// TIA Portal V17 export
// export: Created 2025-03-07T09:17:26.5341874Z, ExportSetting WithDefaults, DisplayName Totally Integrated Automation Portal, DisplayVersion V17 Update 8, DisplayName TIA Portal Openness, DisplayVersion V17 Update 8, DisplayName TIA Portal Version Control Interface, DisplayVersion V17, DisplayName SINAMICS Startdrive Advanced, DisplayVersion V17 SP2, DisplayName SINAMICS Startdrive G110M, G120, G120C, G120D, G120P, G115D, DisplayVersion V17 SP2, DisplayName SINAMICS Startdrive G130, G150, S120, S150, SINAMICS MV, S210, DisplayVersion V17 SP2, DisplayName STEP 7 Professional, DisplayVersion V17 Update 8, DisplayName SINUMERIK ONE STEP 7 Toolbox, DisplayVersion V17 Update 12, DisplayName SINUMERIK 840D sl STEP 7 Toolbox, DisplayVersion V17 Update 12, DisplayName STEP 7 Safety, DisplayVersion V17 Update 6, DisplayName WinCC Advanced, DisplayVersion V17 Update 8
FUNCTION "FC365_NCK_M_CH7_UNIT_2_STA_4" : Void   // FC365, LAD
TITLE = Channel 1 data
{ S7_Optimized_Access := 'FALSE' }
AUTHOR : ETXETAR
VERSION : 1.0
// stored: AutoNumber false, IsIECCheckEnabled false, SetENOAutomatically false, UDAEnableTagReadback false
   VAR_TEMP
      auxm3 : Bool;
      auxm5 : Bool;
   END_VAR
   VAR_TEMP   // added for the SCL form of the ladder/FBD networks
      _w1 : Bool;
      _w2 : Bool;
   END_VAR
BEGIN

REGION Network 1: CALL FB331 M CODE EXTENDED CH4 / M CODE EXTENDED CHANNEL 2
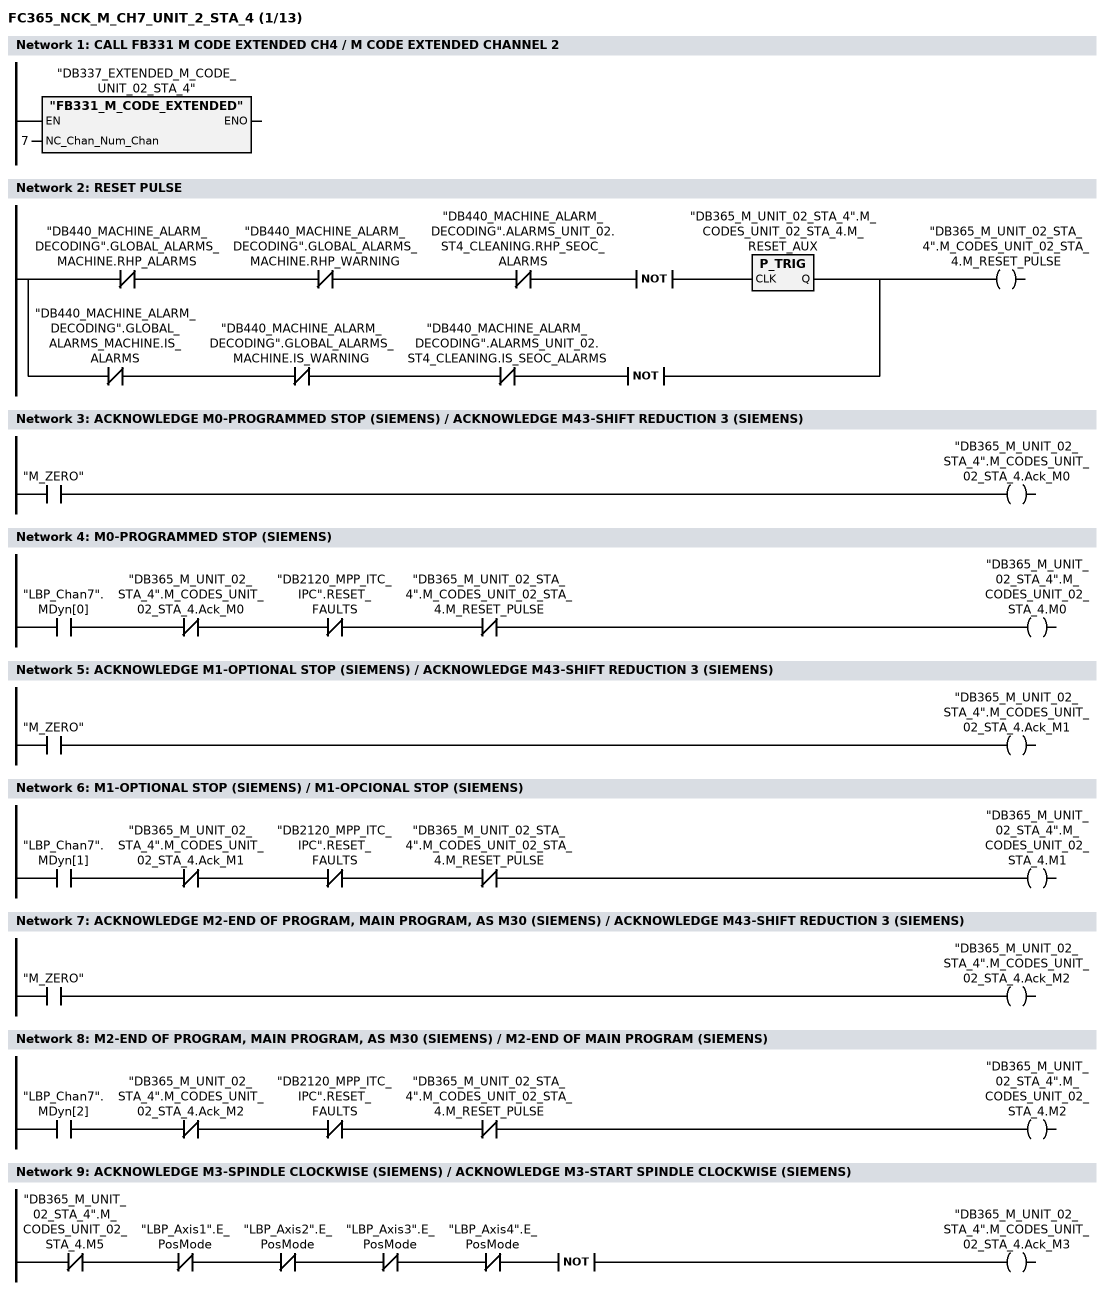
   RUNG wire#powerrail
      "DB337_EXTENDED_M_CODE_UNIT_02_STA_4"(NC_Chan_Num_Chan := 7)
   END_RUNG
   // the same network as SCL:
   "DB337_EXTENDED_M_CODE_UNIT_02_STA_4"(NC_Chan_Num_Chan := 7);   // "FB331_M_CODE_EXTENDED"
END_REGION

REGION Network 2: RESET PULSE
   RUNG wire#powerrail
      I_Contact( "DB440_MACHINE_ALARM_DECODING".GLOBAL_ALARMS_MACHINE.RHP_ALARMS )
      I_Contact( "DB440_MACHINE_ALARM_DECODING".GLOBAL_ALARMS_MACHINE.RHP_WARNING )
      I_Contact( "DB440_MACHINE_ALARM_DECODING".ALARMS_UNIT_02.ST4_CLEANING.RHP_SEOC_ALARMS )
      Not()
      P_Trig( "DB365_M_UNIT_02_STA_4".M_CODES_UNIT_02_STA_4.M_RESET_AUX )
      wire#w1
      Coil( "DB365_M_UNIT_02_STA_4".M_CODES_UNIT_02_STA_4.M_RESET_PULSE )
   END_RUNG
   RUNG wire#powerrail
      I_Contact( "DB440_MACHINE_ALARM_DECODING".GLOBAL_ALARMS_MACHINE.IS_ALARMS )
      I_Contact( "DB440_MACHINE_ALARM_DECODING".GLOBAL_ALARMS_MACHINE.IS_WARNING )
      I_Contact( "DB440_MACHINE_ALARM_DECODING".ALARMS_UNIT_02.ST4_CLEANING.IS_SEOC_ALARMS )
      Not()
   END_RUNG wire#w1
   // the same network as SCL:
   #_w1 := NOT (NOT "DB440_MACHINE_ALARM_DECODING".GLOBAL_ALARMS_MACHINE.RHP_ALARMS AND NOT "DB440_MACHINE_ALARM_DECODING".GLOBAL_ALARMS_MACHINE.RHP_WARNING AND NOT "DB440_MACHINE_ALARM_DECODING".ALARMS_UNIT_02.ST4_CLEANING.RHP_SEOC_ALARMS);
   #_w2 := #_w1 AND NOT "DB365_M_UNIT_02_STA_4".M_CODES_UNIT_02_STA_4.M_RESET_AUX;   // rising edge
   "DB365_M_UNIT_02_STA_4".M_CODES_UNIT_02_STA_4.M_RESET_AUX := #_w1;
   "DB365_M_UNIT_02_STA_4".M_CODES_UNIT_02_STA_4.M_RESET_PULSE := #_w2 OR NOT (NOT "DB440_MACHINE_ALARM_DECODING".GLOBAL_ALARMS_MACHINE.IS_ALARMS AND NOT "DB440_MACHINE_ALARM_DECODING".GLOBAL_ALARMS_MACHINE.IS_WARNING AND NOT "DB440_MACHINE_ALARM_DECODING".ALARMS_UNIT_02.ST4_CLEANING.IS_SEOC_ALARMS);
END_REGION

REGION Network 3: ACKNOWLEDGE M0-PROGRAMMED STOP (SIEMENS) / ACKNOWLEDGE M43-SHIFT REDUCTION 3 (SIEMENS)
   RUNG wire#powerrail
      Contact( "M_ZERO" )
      Coil( "DB365_M_UNIT_02_STA_4".M_CODES_UNIT_02_STA_4.Ack_M0 )
   END_RUNG
   // the same network as SCL:
   "DB365_M_UNIT_02_STA_4".M_CODES_UNIT_02_STA_4.Ack_M0 := "M_ZERO";
END_REGION

REGION Network 4: M0-PROGRAMMED STOP (SIEMENS)
   RUNG wire#powerrail
      Contact( "LBP_Chan7".MDyn[0] )
      I_Contact( "DB365_M_UNIT_02_STA_4".M_CODES_UNIT_02_STA_4.Ack_M0 )
      I_Contact( "DB2120_MPP_ITC_IPC".RESET_FAULTS )
      I_Contact( "DB365_M_UNIT_02_STA_4".M_CODES_UNIT_02_STA_4.M_RESET_PULSE )
      Coil( "DB365_M_UNIT_02_STA_4".M_CODES_UNIT_02_STA_4.M0 )
   END_RUNG
   // the same network as SCL:
   "DB365_M_UNIT_02_STA_4".M_CODES_UNIT_02_STA_4.M0 := "LBP_Chan7".MDyn[0] AND NOT "DB365_M_UNIT_02_STA_4".M_CODES_UNIT_02_STA_4.Ack_M0 AND NOT "DB2120_MPP_ITC_IPC".RESET_FAULTS AND NOT "DB365_M_UNIT_02_STA_4".M_CODES_UNIT_02_STA_4.M_RESET_PULSE;
END_REGION

REGION Network 5: ACKNOWLEDGE M1-OPTIONAL STOP (SIEMENS) / ACKNOWLEDGE M43-SHIFT REDUCTION 3 (SIEMENS)
   RUNG wire#powerrail
      Contact( "M_ZERO" )
      Coil( "DB365_M_UNIT_02_STA_4".M_CODES_UNIT_02_STA_4.Ack_M1 )
   END_RUNG
   // the same network as SCL:
   "DB365_M_UNIT_02_STA_4".M_CODES_UNIT_02_STA_4.Ack_M1 := "M_ZERO";
END_REGION

REGION Network 6: M1-OPTIONAL STOP (SIEMENS) / M1-OPCIONAL STOP (SIEMENS)
   RUNG wire#powerrail
      Contact( "LBP_Chan7".MDyn[1] )
      I_Contact( "DB365_M_UNIT_02_STA_4".M_CODES_UNIT_02_STA_4.Ack_M1 )
      I_Contact( "DB2120_MPP_ITC_IPC".RESET_FAULTS )
      I_Contact( "DB365_M_UNIT_02_STA_4".M_CODES_UNIT_02_STA_4.M_RESET_PULSE )
      Coil( "DB365_M_UNIT_02_STA_4".M_CODES_UNIT_02_STA_4.M1 )
   END_RUNG
   // the same network as SCL:
   "DB365_M_UNIT_02_STA_4".M_CODES_UNIT_02_STA_4.M1 := "LBP_Chan7".MDyn[1] AND NOT "DB365_M_UNIT_02_STA_4".M_CODES_UNIT_02_STA_4.Ack_M1 AND NOT "DB2120_MPP_ITC_IPC".RESET_FAULTS AND NOT "DB365_M_UNIT_02_STA_4".M_CODES_UNIT_02_STA_4.M_RESET_PULSE;
END_REGION

REGION Network 7: ACKNOWLEDGE M2-END OF PROGRAM, MAIN PROGRAM, AS M30 (SIEMENS) / ACKNOWLEDGE M43-SHIFT REDUCTION 3 (SIEMENS)
   RUNG wire#powerrail
      Contact( "M_ZERO" )
      Coil( "DB365_M_UNIT_02_STA_4".M_CODES_UNIT_02_STA_4.Ack_M2 )
   END_RUNG
   // the same network as SCL:
   "DB365_M_UNIT_02_STA_4".M_CODES_UNIT_02_STA_4.Ack_M2 := "M_ZERO";
END_REGION

REGION Network 8: M2-END OF PROGRAM, MAIN PROGRAM, AS M30 (SIEMENS) / M2-END OF MAIN PROGRAM (SIEMENS)
   RUNG wire#powerrail
      Contact( "LBP_Chan7".MDyn[2] )
      I_Contact( "DB365_M_UNIT_02_STA_4".M_CODES_UNIT_02_STA_4.Ack_M2 )
      I_Contact( "DB2120_MPP_ITC_IPC".RESET_FAULTS )
      I_Contact( "DB365_M_UNIT_02_STA_4".M_CODES_UNIT_02_STA_4.M_RESET_PULSE )
      Coil( "DB365_M_UNIT_02_STA_4".M_CODES_UNIT_02_STA_4.M2 )
   END_RUNG
   // the same network as SCL:
   "DB365_M_UNIT_02_STA_4".M_CODES_UNIT_02_STA_4.M2 := "LBP_Chan7".MDyn[2] AND NOT "DB365_M_UNIT_02_STA_4".M_CODES_UNIT_02_STA_4.Ack_M2 AND NOT "DB2120_MPP_ITC_IPC".RESET_FAULTS AND NOT "DB365_M_UNIT_02_STA_4".M_CODES_UNIT_02_STA_4.M_RESET_PULSE;
END_REGION

REGION Network 9: ACKNOWLEDGE M3-SPINDLE CLOCKWISE (SIEMENS) / ACKNOWLEDGE M3-START SPINDLE CLOCKWISE (SIEMENS)
   RUNG wire#powerrail
      I_Contact( "DB365_M_UNIT_02_STA_4".M_CODES_UNIT_02_STA_4.M5 )
      I_Contact( "LBP_Axis1".E_PosMode )
      I_Contact( "LBP_Axis2".E_PosMode )
      I_Contact( "LBP_Axis3".E_PosMode )
      I_Contact( "LBP_Axis4".E_PosMode )
      Not()
      Coil( "DB365_M_UNIT_02_STA_4".M_CODES_UNIT_02_STA_4.Ack_M3 )
   END_RUNG
   // the same network as SCL:
   "DB365_M_UNIT_02_STA_4".M_CODES_UNIT_02_STA_4.Ack_M3 := NOT (NOT "DB365_M_UNIT_02_STA_4".M_CODES_UNIT_02_STA_4.M5 AND NOT "LBP_Axis1".E_PosMode AND NOT "LBP_Axis2".E_PosMode AND NOT "LBP_Axis3".E_PosMode AND NOT "LBP_Axis4".E_PosMode);
END_REGION

REGION Network 10: M3-SPINDLE CLOCKWISE AUXILIARY (SIEMENS) / Extended address M function 1 (16 bit INT)
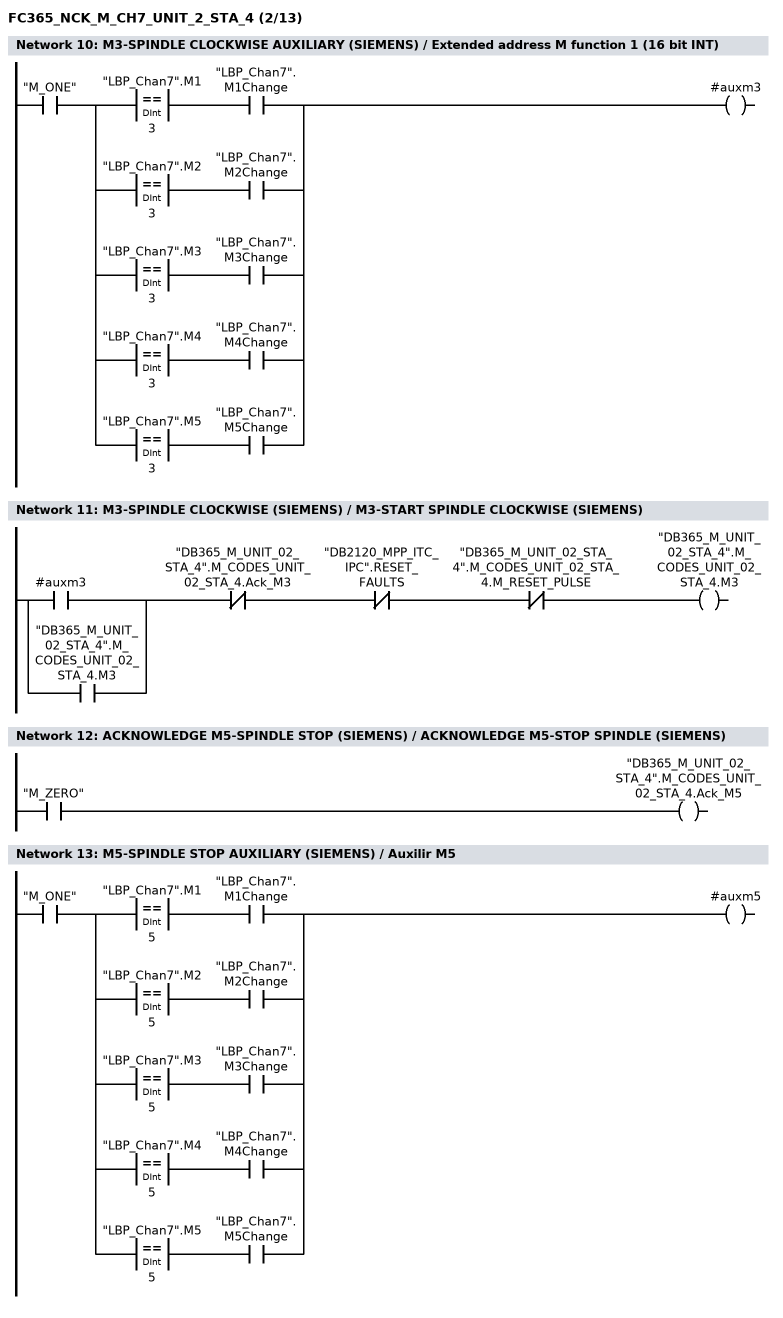
   RUNG wire#powerrail
      Contact( "M_ONE" )
      wire#w1
      { S7_Templates := "SrcType := DInt" } EQ_Contact(in1 := "LBP_Chan7".M1, in2 := 3)
      Contact( "LBP_Chan7".M1Change )
      wire#w2
      Coil( #auxm3 )
   END_RUNG
   RUNG wire#w1
      { S7_Templates := "SrcType := DInt" } EQ_Contact(in1 := "LBP_Chan7".M2, in2 := 3)
      Contact( "LBP_Chan7".M2Change )
   END_RUNG wire#w2
   RUNG wire#w1
      { S7_Templates := "SrcType := DInt" } EQ_Contact(in1 := "LBP_Chan7".M3, in2 := 3)
      Contact( "LBP_Chan7".M3Change )
   END_RUNG wire#w2
   RUNG wire#w1
      { S7_Templates := "SrcType := DInt" } EQ_Contact(in1 := "LBP_Chan7".M4, in2 := 3)
      Contact( "LBP_Chan7".M4Change )
   END_RUNG wire#w2
   RUNG wire#w1
      { S7_Templates := "SrcType := DInt" } EQ_Contact(in1 := "LBP_Chan7".M5, in2 := 3)
      Contact( "LBP_Chan7".M5Change )
   END_RUNG wire#w2
   // the same network as SCL:
   #auxm3 := "M_ONE" AND ((("LBP_Chan7".M1 = 3) AND "LBP_Chan7".M1Change) OR (("LBP_Chan7".M2 = 3) AND "LBP_Chan7".M2Change) OR (("LBP_Chan7".M3 = 3) AND "LBP_Chan7".M3Change) OR (("LBP_Chan7".M4 = 3) AND "LBP_Chan7".M4Change) OR (("LBP_Chan7".M5 = 3) AND "LBP_Chan7".M5Change));
END_REGION

REGION Network 11: M3-SPINDLE CLOCKWISE (SIEMENS) / M3-START SPINDLE CLOCKWISE (SIEMENS)
   RUNG wire#powerrail
      Contact( #auxm3 )
      wire#w1
      I_Contact( "DB365_M_UNIT_02_STA_4".M_CODES_UNIT_02_STA_4.Ack_M3 )
      I_Contact( "DB2120_MPP_ITC_IPC".RESET_FAULTS )
      I_Contact( "DB365_M_UNIT_02_STA_4".M_CODES_UNIT_02_STA_4.M_RESET_PULSE )
      Coil( "DB365_M_UNIT_02_STA_4".M_CODES_UNIT_02_STA_4.M3 )
   END_RUNG
   RUNG wire#powerrail
      Contact( "DB365_M_UNIT_02_STA_4".M_CODES_UNIT_02_STA_4.M3 )
   END_RUNG wire#w1
   // the same network as SCL:
   "DB365_M_UNIT_02_STA_4".M_CODES_UNIT_02_STA_4.M3 := (#auxm3 OR "DB365_M_UNIT_02_STA_4".M_CODES_UNIT_02_STA_4.M3) AND NOT "DB365_M_UNIT_02_STA_4".M_CODES_UNIT_02_STA_4.Ack_M3 AND NOT "DB2120_MPP_ITC_IPC".RESET_FAULTS AND NOT "DB365_M_UNIT_02_STA_4".M_CODES_UNIT_02_STA_4.M_RESET_PULSE;
END_REGION

REGION Network 12: ACKNOWLEDGE M5-SPINDLE STOP (SIEMENS) / ACKNOWLEDGE M5-STOP SPINDLE (SIEMENS)
   RUNG wire#powerrail
      Contact( "M_ZERO" )
      Coil( "DB365_M_UNIT_02_STA_4".M_CODES_UNIT_02_STA_4.Ack_M5 )
   END_RUNG
   // the same network as SCL:
   "DB365_M_UNIT_02_STA_4".M_CODES_UNIT_02_STA_4.Ack_M5 := "M_ZERO";
END_REGION

REGION Network 13: M5-SPINDLE STOP AUXILIARY (SIEMENS) / Auxilir M5
   RUNG wire#powerrail
      Contact( "M_ONE" )
      wire#w1
      { S7_Templates := "SrcType := DInt" } EQ_Contact(in1 := "LBP_Chan7".M1, in2 := 5)
      Contact( "LBP_Chan7".M1Change )
      wire#w2
      Coil( #auxm5 )
   END_RUNG
   RUNG wire#w1
      { S7_Templates := "SrcType := DInt" } EQ_Contact(in1 := "LBP_Chan7".M2, in2 := 5)
      Contact( "LBP_Chan7".M2Change )
   END_RUNG wire#w2
   RUNG wire#w1
      { S7_Templates := "SrcType := DInt" } EQ_Contact(in1 := "LBP_Chan7".M3, in2 := 5)
      Contact( "LBP_Chan7".M3Change )
   END_RUNG wire#w2
   RUNG wire#w1
      { S7_Templates := "SrcType := DInt" } EQ_Contact(in1 := "LBP_Chan7".M4, in2 := 5)
      Contact( "LBP_Chan7".M4Change )
   END_RUNG wire#w2
   RUNG wire#w1
      { S7_Templates := "SrcType := DInt" } EQ_Contact(in1 := "LBP_Chan7".M5, in2 := 5)
      Contact( "LBP_Chan7".M5Change )
   END_RUNG wire#w2
   // the same network as SCL:
   #auxm5 := "M_ONE" AND ((("LBP_Chan7".M1 = 5) AND "LBP_Chan7".M1Change) OR (("LBP_Chan7".M2 = 5) AND "LBP_Chan7".M2Change) OR (("LBP_Chan7".M3 = 5) AND "LBP_Chan7".M3Change) OR (("LBP_Chan7".M4 = 5) AND "LBP_Chan7".M4Change) OR (("LBP_Chan7".M5 = 5) AND "LBP_Chan7".M5Change));
END_REGION

REGION Network 14: M5-SPINDLE STOP (SIEMENS) / M5-STOP SPINDLE (SIEMENS)
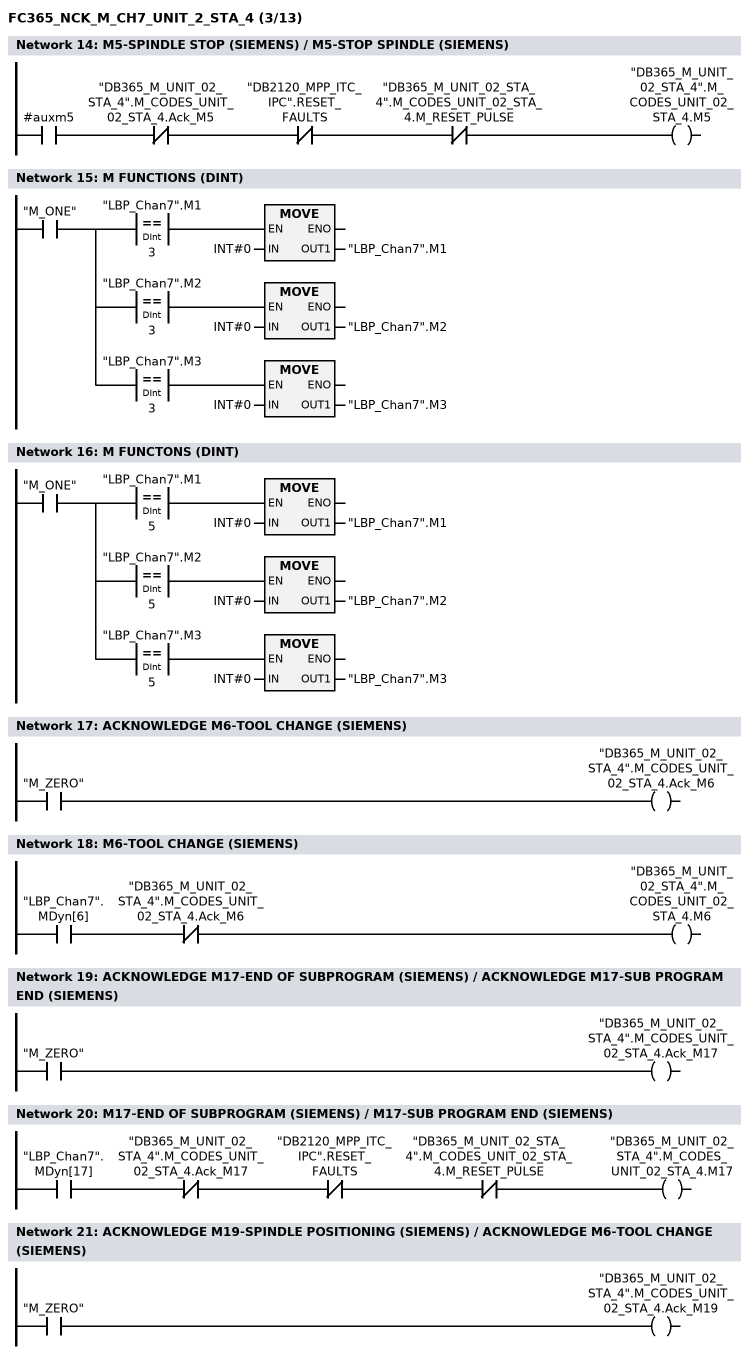
   RUNG wire#powerrail
      Contact( #auxm5 )
      I_Contact( "DB365_M_UNIT_02_STA_4".M_CODES_UNIT_02_STA_4.Ack_M5 )
      I_Contact( "DB2120_MPP_ITC_IPC".RESET_FAULTS )
      I_Contact( "DB365_M_UNIT_02_STA_4".M_CODES_UNIT_02_STA_4.M_RESET_PULSE )
      Coil( "DB365_M_UNIT_02_STA_4".M_CODES_UNIT_02_STA_4.M5 )
   END_RUNG
   // the same network as SCL:
   "DB365_M_UNIT_02_STA_4".M_CODES_UNIT_02_STA_4.M5 := #auxm5 AND NOT "DB365_M_UNIT_02_STA_4".M_CODES_UNIT_02_STA_4.Ack_M5 AND NOT "DB2120_MPP_ITC_IPC".RESET_FAULTS AND NOT "DB365_M_UNIT_02_STA_4".M_CODES_UNIT_02_STA_4.M_RESET_PULSE;
END_REGION

REGION Network 15: M FUNCTIONS (DINT)
   RUNG wire#powerrail
      Contact( "M_ONE" )
      wire#w1
      { S7_Templates := "SrcType := DInt" } EQ_Contact(in1 := "LBP_Chan7".M1, in2 := 3)
      { S7_GenerateENO := "TRUE" } Move(in := INT#0, out1 => "LBP_Chan7".M1)
   END_RUNG
   RUNG wire#w1
      { S7_Templates := "SrcType := DInt" } EQ_Contact(in1 := "LBP_Chan7".M2, in2 := 3)
      { S7_GenerateENO := "TRUE" } Move(in := INT#0, out1 => "LBP_Chan7".M2)
   END_RUNG
   RUNG wire#w1
      { S7_Templates := "SrcType := DInt" } EQ_Contact(in1 := "LBP_Chan7".M3, in2 := 3)
      { S7_GenerateENO := "TRUE" } Move(in := INT#0, out1 => "LBP_Chan7".M3)
   END_RUNG
   // the same network as SCL:
   IF "M_ONE" AND ("LBP_Chan7".M1 = 3) THEN "LBP_Chan7".M1 := INT#0; END_IF;
   IF "M_ONE" AND ("LBP_Chan7".M2 = 3) THEN "LBP_Chan7".M2 := INT#0; END_IF;
   IF "M_ONE" AND ("LBP_Chan7".M3 = 3) THEN "LBP_Chan7".M3 := INT#0; END_IF;
END_REGION

REGION Network 16: M FUNCTONS (DINT)
   RUNG wire#powerrail
      Contact( "M_ONE" )
      wire#w1
      { S7_Templates := "SrcType := DInt" } EQ_Contact(in1 := "LBP_Chan7".M1, in2 := 5)
      { S7_GenerateENO := "TRUE" } Move(in := INT#0, out1 => "LBP_Chan7".M1)
   END_RUNG
   RUNG wire#w1
      { S7_Templates := "SrcType := DInt" } EQ_Contact(in1 := "LBP_Chan7".M2, in2 := 5)
      { S7_GenerateENO := "TRUE" } Move(in := INT#0, out1 => "LBP_Chan7".M2)
   END_RUNG
   RUNG wire#w1
      { S7_Templates := "SrcType := DInt" } EQ_Contact(in1 := "LBP_Chan7".M3, in2 := 5)
      { S7_GenerateENO := "TRUE" } Move(in := INT#0, out1 => "LBP_Chan7".M3)
   END_RUNG
   // the same network as SCL:
   IF "M_ONE" AND ("LBP_Chan7".M1 = 5) THEN "LBP_Chan7".M1 := INT#0; END_IF;
   IF "M_ONE" AND ("LBP_Chan7".M2 = 5) THEN "LBP_Chan7".M2 := INT#0; END_IF;
   IF "M_ONE" AND ("LBP_Chan7".M3 = 5) THEN "LBP_Chan7".M3 := INT#0; END_IF;
END_REGION

REGION Network 17: ACKNOWLEDGE M6-TOOL CHANGE (SIEMENS)
   RUNG wire#powerrail
      Contact( "M_ZERO" )
      Coil( "DB365_M_UNIT_02_STA_4".M_CODES_UNIT_02_STA_4.Ack_M6 )
   END_RUNG
   // the same network as SCL:
   "DB365_M_UNIT_02_STA_4".M_CODES_UNIT_02_STA_4.Ack_M6 := "M_ZERO";
END_REGION

REGION Network 18: M6-TOOL CHANGE (SIEMENS)
   RUNG wire#powerrail
      Contact( "LBP_Chan7".MDyn[6] )
      I_Contact( "DB365_M_UNIT_02_STA_4".M_CODES_UNIT_02_STA_4.Ack_M6 )
      Coil( "DB365_M_UNIT_02_STA_4".M_CODES_UNIT_02_STA_4.M6 )
   END_RUNG
   // the same network as SCL:
   "DB365_M_UNIT_02_STA_4".M_CODES_UNIT_02_STA_4.M6 := "LBP_Chan7".MDyn[6] AND NOT "DB365_M_UNIT_02_STA_4".M_CODES_UNIT_02_STA_4.Ack_M6;
END_REGION

REGION Network 19: ACKNOWLEDGE M17-END OF SUBPROGRAM (SIEMENS) / ACKNOWLEDGE M17-SUB PROGRAM END (SIEMENS)
   RUNG wire#powerrail
      Contact( "M_ZERO" )
      Coil( "DB365_M_UNIT_02_STA_4".M_CODES_UNIT_02_STA_4.Ack_M17 )
   END_RUNG
   // the same network as SCL:
   "DB365_M_UNIT_02_STA_4".M_CODES_UNIT_02_STA_4.Ack_M17 := "M_ZERO";
END_REGION

REGION Network 20: M17-END OF SUBPROGRAM (SIEMENS) / M17-SUB PROGRAM END (SIEMENS)
   RUNG wire#powerrail
      Contact( "LBP_Chan7".MDyn[17] )
      I_Contact( "DB365_M_UNIT_02_STA_4".M_CODES_UNIT_02_STA_4.Ack_M17 )
      I_Contact( "DB2120_MPP_ITC_IPC".RESET_FAULTS )
      I_Contact( "DB365_M_UNIT_02_STA_4".M_CODES_UNIT_02_STA_4.M_RESET_PULSE )
      Coil( "DB365_M_UNIT_02_STA_4".M_CODES_UNIT_02_STA_4.M17 )
   END_RUNG
   // the same network as SCL:
   "DB365_M_UNIT_02_STA_4".M_CODES_UNIT_02_STA_4.M17 := "LBP_Chan7".MDyn[17] AND NOT "DB365_M_UNIT_02_STA_4".M_CODES_UNIT_02_STA_4.Ack_M17 AND NOT "DB2120_MPP_ITC_IPC".RESET_FAULTS AND NOT "DB365_M_UNIT_02_STA_4".M_CODES_UNIT_02_STA_4.M_RESET_PULSE;
END_REGION

REGION Network 21: ACKNOWLEDGE M19-SPINDLE POSITIONING (SIEMENS) / ACKNOWLEDGE M6-TOOL CHANGE (SIEMENS)
   RUNG wire#powerrail
      Contact( "M_ZERO" )
      Coil( "DB365_M_UNIT_02_STA_4".M_CODES_UNIT_02_STA_4.Ack_M19 )
   END_RUNG
   // the same network as SCL:
   "DB365_M_UNIT_02_STA_4".M_CODES_UNIT_02_STA_4.Ack_M19 := "M_ZERO";
END_REGION

REGION Network 22: M19-SPINDLE POSITIONING (SIEMENS) / M6-TOOL CHANGE (SIEMENS)
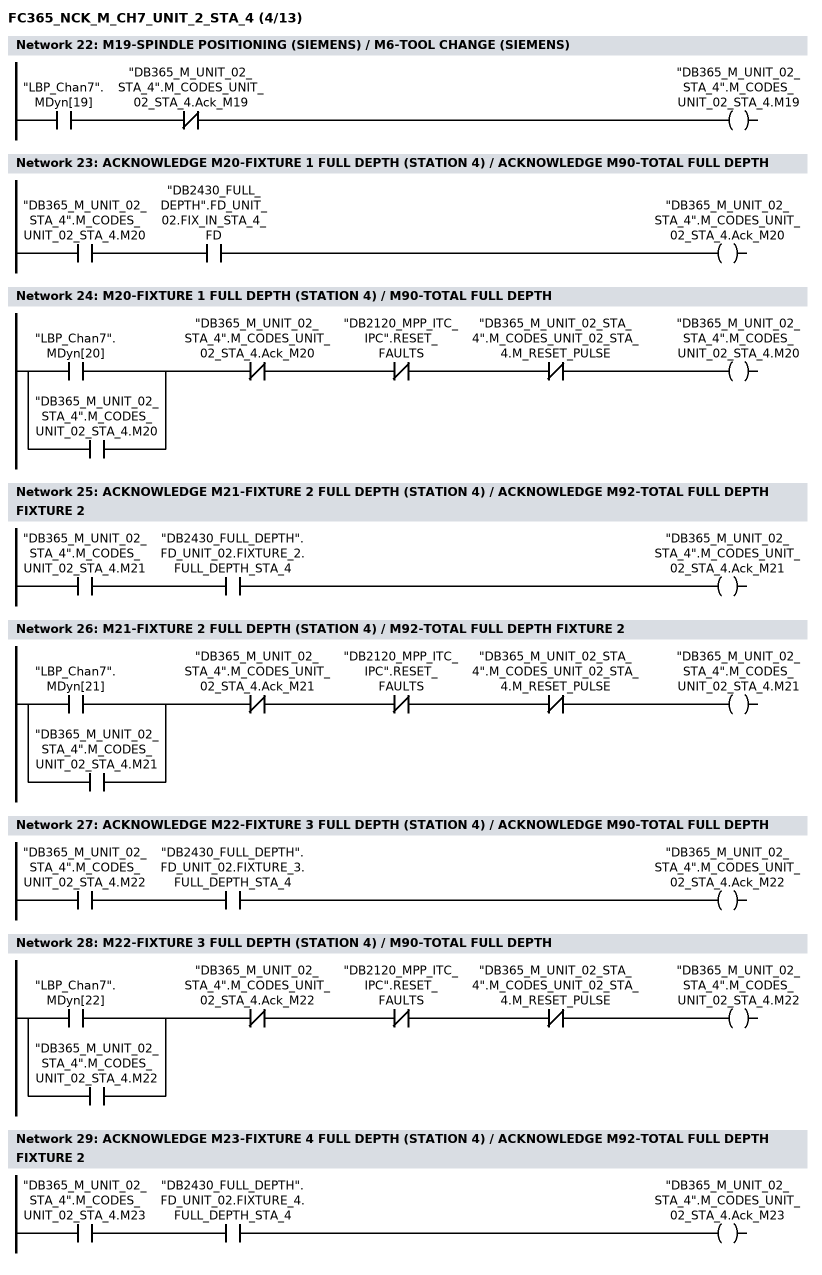
   RUNG wire#powerrail
      Contact( "LBP_Chan7".MDyn[19] )
      I_Contact( "DB365_M_UNIT_02_STA_4".M_CODES_UNIT_02_STA_4.Ack_M19 )
      Coil( "DB365_M_UNIT_02_STA_4".M_CODES_UNIT_02_STA_4.M19 )
   END_RUNG
   // the same network as SCL:
   "DB365_M_UNIT_02_STA_4".M_CODES_UNIT_02_STA_4.M19 := "LBP_Chan7".MDyn[19] AND NOT "DB365_M_UNIT_02_STA_4".M_CODES_UNIT_02_STA_4.Ack_M19;
END_REGION

REGION Network 23: ACKNOWLEDGE M20-FIXTURE 1 FULL DEPTH (STATION 4) / ACKNOWLEDGE M90-TOTAL FULL DEPTH
   RUNG wire#powerrail
      Contact( "DB365_M_UNIT_02_STA_4".M_CODES_UNIT_02_STA_4.M20 )
      Contact( "DB2430_FULL_DEPTH".FD_UNIT_02.FIX_IN_STA_4_FD )
      Coil( "DB365_M_UNIT_02_STA_4".M_CODES_UNIT_02_STA_4.Ack_M20 )
   END_RUNG
   // the same network as SCL:
   "DB365_M_UNIT_02_STA_4".M_CODES_UNIT_02_STA_4.Ack_M20 := "DB365_M_UNIT_02_STA_4".M_CODES_UNIT_02_STA_4.M20 AND "DB2430_FULL_DEPTH".FD_UNIT_02.FIX_IN_STA_4_FD;
END_REGION

REGION Network 24: M20-FIXTURE 1 FULL DEPTH (STATION 4) / M90-TOTAL FULL DEPTH
   RUNG wire#powerrail
      Contact( "LBP_Chan7".MDyn[20] )
      wire#w1
      I_Contact( "DB365_M_UNIT_02_STA_4".M_CODES_UNIT_02_STA_4.Ack_M20 )
      I_Contact( "DB2120_MPP_ITC_IPC".RESET_FAULTS )
      I_Contact( "DB365_M_UNIT_02_STA_4".M_CODES_UNIT_02_STA_4.M_RESET_PULSE )
      Coil( "DB365_M_UNIT_02_STA_4".M_CODES_UNIT_02_STA_4.M20 )
   END_RUNG
   RUNG wire#powerrail
      Contact( "DB365_M_UNIT_02_STA_4".M_CODES_UNIT_02_STA_4.M20 )
   END_RUNG wire#w1
   // the same network as SCL:
   "DB365_M_UNIT_02_STA_4".M_CODES_UNIT_02_STA_4.M20 := ("LBP_Chan7".MDyn[20] OR "DB365_M_UNIT_02_STA_4".M_CODES_UNIT_02_STA_4.M20) AND NOT "DB365_M_UNIT_02_STA_4".M_CODES_UNIT_02_STA_4.Ack_M20 AND NOT "DB2120_MPP_ITC_IPC".RESET_FAULTS AND NOT "DB365_M_UNIT_02_STA_4".M_CODES_UNIT_02_STA_4.M_RESET_PULSE;
END_REGION

REGION Network 25: ACKNOWLEDGE M21-FIXTURE 2 FULL DEPTH (STATION 4) / ACKNOWLEDGE M92-TOTAL FULL DEPTH FIXTURE 2
   RUNG wire#powerrail
      Contact( "DB365_M_UNIT_02_STA_4".M_CODES_UNIT_02_STA_4.M21 )
      Contact( "DB2430_FULL_DEPTH".FD_UNIT_02.FIXTURE_2.FULL_DEPTH_STA_4 )
      Coil( "DB365_M_UNIT_02_STA_4".M_CODES_UNIT_02_STA_4.Ack_M21 )
   END_RUNG
   // the same network as SCL:
   "DB365_M_UNIT_02_STA_4".M_CODES_UNIT_02_STA_4.Ack_M21 := "DB365_M_UNIT_02_STA_4".M_CODES_UNIT_02_STA_4.M21 AND "DB2430_FULL_DEPTH".FD_UNIT_02.FIXTURE_2.FULL_DEPTH_STA_4;
END_REGION

REGION Network 26: M21-FIXTURE 2 FULL DEPTH (STATION 4) / M92-TOTAL FULL DEPTH FIXTURE 2
   RUNG wire#powerrail
      Contact( "LBP_Chan7".MDyn[21] )
      wire#w1
      I_Contact( "DB365_M_UNIT_02_STA_4".M_CODES_UNIT_02_STA_4.Ack_M21 )
      I_Contact( "DB2120_MPP_ITC_IPC".RESET_FAULTS )
      I_Contact( "DB365_M_UNIT_02_STA_4".M_CODES_UNIT_02_STA_4.M_RESET_PULSE )
      Coil( "DB365_M_UNIT_02_STA_4".M_CODES_UNIT_02_STA_4.M21 )
   END_RUNG
   RUNG wire#powerrail
      Contact( "DB365_M_UNIT_02_STA_4".M_CODES_UNIT_02_STA_4.M21 )
   END_RUNG wire#w1
   // the same network as SCL:
   "DB365_M_UNIT_02_STA_4".M_CODES_UNIT_02_STA_4.M21 := ("LBP_Chan7".MDyn[21] OR "DB365_M_UNIT_02_STA_4".M_CODES_UNIT_02_STA_4.M21) AND NOT "DB365_M_UNIT_02_STA_4".M_CODES_UNIT_02_STA_4.Ack_M21 AND NOT "DB2120_MPP_ITC_IPC".RESET_FAULTS AND NOT "DB365_M_UNIT_02_STA_4".M_CODES_UNIT_02_STA_4.M_RESET_PULSE;
END_REGION

REGION Network 27: ACKNOWLEDGE M22-FIXTURE 3 FULL DEPTH (STATION 4) / ACKNOWLEDGE M90-TOTAL FULL DEPTH
   RUNG wire#powerrail
      Contact( "DB365_M_UNIT_02_STA_4".M_CODES_UNIT_02_STA_4.M22 )
      Contact( "DB2430_FULL_DEPTH".FD_UNIT_02.FIXTURE_3.FULL_DEPTH_STA_4 )
      Coil( "DB365_M_UNIT_02_STA_4".M_CODES_UNIT_02_STA_4.Ack_M22 )
   END_RUNG
   // the same network as SCL:
   "DB365_M_UNIT_02_STA_4".M_CODES_UNIT_02_STA_4.Ack_M22 := "DB365_M_UNIT_02_STA_4".M_CODES_UNIT_02_STA_4.M22 AND "DB2430_FULL_DEPTH".FD_UNIT_02.FIXTURE_3.FULL_DEPTH_STA_4;
END_REGION

REGION Network 28: M22-FIXTURE 3 FULL DEPTH (STATION 4) / M90-TOTAL FULL DEPTH
   RUNG wire#powerrail
      Contact( "LBP_Chan7".MDyn[22] )
      wire#w1
      I_Contact( "DB365_M_UNIT_02_STA_4".M_CODES_UNIT_02_STA_4.Ack_M22 )
      I_Contact( "DB2120_MPP_ITC_IPC".RESET_FAULTS )
      I_Contact( "DB365_M_UNIT_02_STA_4".M_CODES_UNIT_02_STA_4.M_RESET_PULSE )
      Coil( "DB365_M_UNIT_02_STA_4".M_CODES_UNIT_02_STA_4.M22 )
   END_RUNG
   RUNG wire#powerrail
      Contact( "DB365_M_UNIT_02_STA_4".M_CODES_UNIT_02_STA_4.M22 )
   END_RUNG wire#w1
   // the same network as SCL:
   "DB365_M_UNIT_02_STA_4".M_CODES_UNIT_02_STA_4.M22 := ("LBP_Chan7".MDyn[22] OR "DB365_M_UNIT_02_STA_4".M_CODES_UNIT_02_STA_4.M22) AND NOT "DB365_M_UNIT_02_STA_4".M_CODES_UNIT_02_STA_4.Ack_M22 AND NOT "DB2120_MPP_ITC_IPC".RESET_FAULTS AND NOT "DB365_M_UNIT_02_STA_4".M_CODES_UNIT_02_STA_4.M_RESET_PULSE;
END_REGION

REGION Network 29: ACKNOWLEDGE M23-FIXTURE 4 FULL DEPTH (STATION 4) / ACKNOWLEDGE M92-TOTAL FULL DEPTH FIXTURE 2
   RUNG wire#powerrail
      Contact( "DB365_M_UNIT_02_STA_4".M_CODES_UNIT_02_STA_4.M23 )
      Contact( "DB2430_FULL_DEPTH".FD_UNIT_02.FIXTURE_4.FULL_DEPTH_STA_4 )
      Coil( "DB365_M_UNIT_02_STA_4".M_CODES_UNIT_02_STA_4.Ack_M23 )
   END_RUNG
   // the same network as SCL:
   "DB365_M_UNIT_02_STA_4".M_CODES_UNIT_02_STA_4.Ack_M23 := "DB365_M_UNIT_02_STA_4".M_CODES_UNIT_02_STA_4.M23 AND "DB2430_FULL_DEPTH".FD_UNIT_02.FIXTURE_4.FULL_DEPTH_STA_4;
END_REGION

REGION Network 30: M23-FIXTURE 4 FULL DEPTH (STATION 4) / M92-TOTAL FULL DEPTH FIXTURE 2
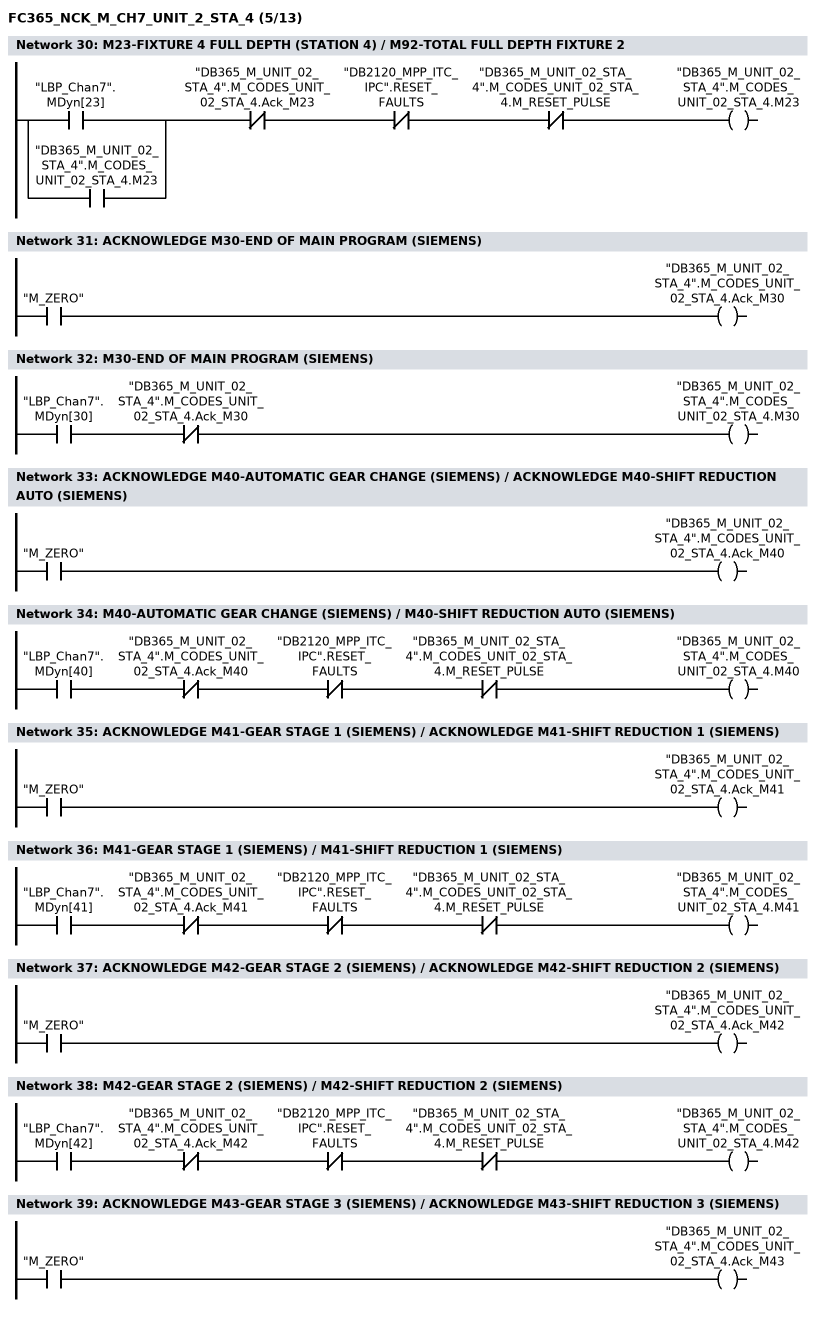
   RUNG wire#powerrail
      Contact( "LBP_Chan7".MDyn[23] )
      wire#w1
      I_Contact( "DB365_M_UNIT_02_STA_4".M_CODES_UNIT_02_STA_4.Ack_M23 )
      I_Contact( "DB2120_MPP_ITC_IPC".RESET_FAULTS )
      I_Contact( "DB365_M_UNIT_02_STA_4".M_CODES_UNIT_02_STA_4.M_RESET_PULSE )
      Coil( "DB365_M_UNIT_02_STA_4".M_CODES_UNIT_02_STA_4.M23 )
   END_RUNG
   RUNG wire#powerrail
      Contact( "DB365_M_UNIT_02_STA_4".M_CODES_UNIT_02_STA_4.M23 )
   END_RUNG wire#w1
   // the same network as SCL:
   "DB365_M_UNIT_02_STA_4".M_CODES_UNIT_02_STA_4.M23 := ("LBP_Chan7".MDyn[23] OR "DB365_M_UNIT_02_STA_4".M_CODES_UNIT_02_STA_4.M23) AND NOT "DB365_M_UNIT_02_STA_4".M_CODES_UNIT_02_STA_4.Ack_M23 AND NOT "DB2120_MPP_ITC_IPC".RESET_FAULTS AND NOT "DB365_M_UNIT_02_STA_4".M_CODES_UNIT_02_STA_4.M_RESET_PULSE;
END_REGION

REGION Network 31: ACKNOWLEDGE M30-END OF MAIN PROGRAM (SIEMENS)
   RUNG wire#powerrail
      Contact( "M_ZERO" )
      Coil( "DB365_M_UNIT_02_STA_4".M_CODES_UNIT_02_STA_4.Ack_M30 )
   END_RUNG
   // the same network as SCL:
   "DB365_M_UNIT_02_STA_4".M_CODES_UNIT_02_STA_4.Ack_M30 := "M_ZERO";
END_REGION

REGION Network 32: M30-END OF MAIN PROGRAM (SIEMENS)
   RUNG wire#powerrail
      Contact( "LBP_Chan7".MDyn[30] )
      I_Contact( "DB365_M_UNIT_02_STA_4".M_CODES_UNIT_02_STA_4.Ack_M30 )
      Coil( "DB365_M_UNIT_02_STA_4".M_CODES_UNIT_02_STA_4.M30 )
   END_RUNG
   // the same network as SCL:
   "DB365_M_UNIT_02_STA_4".M_CODES_UNIT_02_STA_4.M30 := "LBP_Chan7".MDyn[30] AND NOT "DB365_M_UNIT_02_STA_4".M_CODES_UNIT_02_STA_4.Ack_M30;
END_REGION

REGION Network 33: ACKNOWLEDGE M40-AUTOMATIC GEAR CHANGE (SIEMENS) / ACKNOWLEDGE M40-SHIFT REDUCTION AUTO (SIEMENS)
   RUNG wire#powerrail
      Contact( "M_ZERO" )
      Coil( "DB365_M_UNIT_02_STA_4".M_CODES_UNIT_02_STA_4.Ack_M40 )
   END_RUNG
   // the same network as SCL:
   "DB365_M_UNIT_02_STA_4".M_CODES_UNIT_02_STA_4.Ack_M40 := "M_ZERO";
END_REGION

REGION Network 34: M40-AUTOMATIC GEAR CHANGE (SIEMENS) / M40-SHIFT REDUCTION AUTO (SIEMENS)
   RUNG wire#powerrail
      Contact( "LBP_Chan7".MDyn[40] )
      I_Contact( "DB365_M_UNIT_02_STA_4".M_CODES_UNIT_02_STA_4.Ack_M40 )
      I_Contact( "DB2120_MPP_ITC_IPC".RESET_FAULTS )
      I_Contact( "DB365_M_UNIT_02_STA_4".M_CODES_UNIT_02_STA_4.M_RESET_PULSE )
      Coil( "DB365_M_UNIT_02_STA_4".M_CODES_UNIT_02_STA_4.M40 )
   END_RUNG
   // the same network as SCL:
   "DB365_M_UNIT_02_STA_4".M_CODES_UNIT_02_STA_4.M40 := "LBP_Chan7".MDyn[40] AND NOT "DB365_M_UNIT_02_STA_4".M_CODES_UNIT_02_STA_4.Ack_M40 AND NOT "DB2120_MPP_ITC_IPC".RESET_FAULTS AND NOT "DB365_M_UNIT_02_STA_4".M_CODES_UNIT_02_STA_4.M_RESET_PULSE;
END_REGION

REGION Network 35: ACKNOWLEDGE M41-GEAR STAGE 1 (SIEMENS) / ACKNOWLEDGE M41-SHIFT REDUCTION 1 (SIEMENS)
   RUNG wire#powerrail
      Contact( "M_ZERO" )
      Coil( "DB365_M_UNIT_02_STA_4".M_CODES_UNIT_02_STA_4.Ack_M41 )
   END_RUNG
   // the same network as SCL:
   "DB365_M_UNIT_02_STA_4".M_CODES_UNIT_02_STA_4.Ack_M41 := "M_ZERO";
END_REGION

REGION Network 36: M41-GEAR STAGE 1 (SIEMENS) / M41-SHIFT REDUCTION 1 (SIEMENS)
   RUNG wire#powerrail
      Contact( "LBP_Chan7".MDyn[41] )
      I_Contact( "DB365_M_UNIT_02_STA_4".M_CODES_UNIT_02_STA_4.Ack_M41 )
      I_Contact( "DB2120_MPP_ITC_IPC".RESET_FAULTS )
      I_Contact( "DB365_M_UNIT_02_STA_4".M_CODES_UNIT_02_STA_4.M_RESET_PULSE )
      Coil( "DB365_M_UNIT_02_STA_4".M_CODES_UNIT_02_STA_4.M41 )
   END_RUNG
   // the same network as SCL:
   "DB365_M_UNIT_02_STA_4".M_CODES_UNIT_02_STA_4.M41 := "LBP_Chan7".MDyn[41] AND NOT "DB365_M_UNIT_02_STA_4".M_CODES_UNIT_02_STA_4.Ack_M41 AND NOT "DB2120_MPP_ITC_IPC".RESET_FAULTS AND NOT "DB365_M_UNIT_02_STA_4".M_CODES_UNIT_02_STA_4.M_RESET_PULSE;
END_REGION

REGION Network 37: ACKNOWLEDGE M42-GEAR STAGE 2 (SIEMENS) / ACKNOWLEDGE M42-SHIFT REDUCTION 2 (SIEMENS)
   RUNG wire#powerrail
      Contact( "M_ZERO" )
      Coil( "DB365_M_UNIT_02_STA_4".M_CODES_UNIT_02_STA_4.Ack_M42 )
   END_RUNG
   // the same network as SCL:
   "DB365_M_UNIT_02_STA_4".M_CODES_UNIT_02_STA_4.Ack_M42 := "M_ZERO";
END_REGION

REGION Network 38: M42-GEAR STAGE 2 (SIEMENS) / M42-SHIFT REDUCTION 2 (SIEMENS)
   RUNG wire#powerrail
      Contact( "LBP_Chan7".MDyn[42] )
      I_Contact( "DB365_M_UNIT_02_STA_4".M_CODES_UNIT_02_STA_4.Ack_M42 )
      I_Contact( "DB2120_MPP_ITC_IPC".RESET_FAULTS )
      I_Contact( "DB365_M_UNIT_02_STA_4".M_CODES_UNIT_02_STA_4.M_RESET_PULSE )
      Coil( "DB365_M_UNIT_02_STA_4".M_CODES_UNIT_02_STA_4.M42 )
   END_RUNG
   // the same network as SCL:
   "DB365_M_UNIT_02_STA_4".M_CODES_UNIT_02_STA_4.M42 := "LBP_Chan7".MDyn[42] AND NOT "DB365_M_UNIT_02_STA_4".M_CODES_UNIT_02_STA_4.Ack_M42 AND NOT "DB2120_MPP_ITC_IPC".RESET_FAULTS AND NOT "DB365_M_UNIT_02_STA_4".M_CODES_UNIT_02_STA_4.M_RESET_PULSE;
END_REGION

REGION Network 39: ACKNOWLEDGE M43-GEAR STAGE 3 (SIEMENS) / ACKNOWLEDGE M43-SHIFT REDUCTION 3 (SIEMENS)
   RUNG wire#powerrail
      Contact( "M_ZERO" )
      Coil( "DB365_M_UNIT_02_STA_4".M_CODES_UNIT_02_STA_4.Ack_M43 )
   END_RUNG
   // the same network as SCL:
   "DB365_M_UNIT_02_STA_4".M_CODES_UNIT_02_STA_4.Ack_M43 := "M_ZERO";
END_REGION

REGION Network 40: M43-GEAR STAGE 3 (SIEMENS) / M43-SHIFT REDUCTION 3 (SIEMENS)
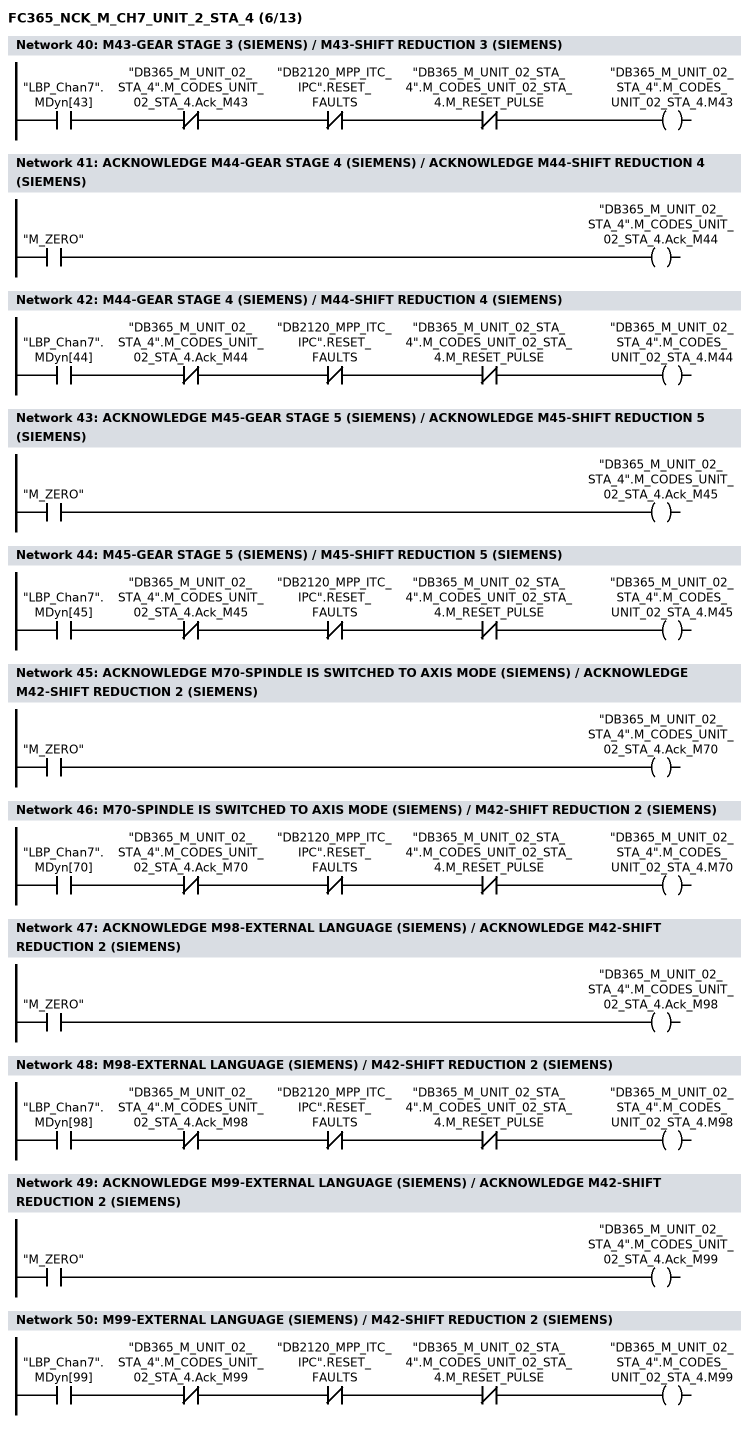
   RUNG wire#powerrail
      Contact( "LBP_Chan7".MDyn[43] )
      I_Contact( "DB365_M_UNIT_02_STA_4".M_CODES_UNIT_02_STA_4.Ack_M43 )
      I_Contact( "DB2120_MPP_ITC_IPC".RESET_FAULTS )
      I_Contact( "DB365_M_UNIT_02_STA_4".M_CODES_UNIT_02_STA_4.M_RESET_PULSE )
      Coil( "DB365_M_UNIT_02_STA_4".M_CODES_UNIT_02_STA_4.M43 )
   END_RUNG
   // the same network as SCL:
   "DB365_M_UNIT_02_STA_4".M_CODES_UNIT_02_STA_4.M43 := "LBP_Chan7".MDyn[43] AND NOT "DB365_M_UNIT_02_STA_4".M_CODES_UNIT_02_STA_4.Ack_M43 AND NOT "DB2120_MPP_ITC_IPC".RESET_FAULTS AND NOT "DB365_M_UNIT_02_STA_4".M_CODES_UNIT_02_STA_4.M_RESET_PULSE;
END_REGION

REGION Network 41: ACKNOWLEDGE M44-GEAR STAGE 4 (SIEMENS) / ACKNOWLEDGE M44-SHIFT REDUCTION 4 (SIEMENS)
   RUNG wire#powerrail
      Contact( "M_ZERO" )
      Coil( "DB365_M_UNIT_02_STA_4".M_CODES_UNIT_02_STA_4.Ack_M44 )
   END_RUNG
   // the same network as SCL:
   "DB365_M_UNIT_02_STA_4".M_CODES_UNIT_02_STA_4.Ack_M44 := "M_ZERO";
END_REGION

REGION Network 42: M44-GEAR STAGE 4 (SIEMENS) / M44-SHIFT REDUCTION 4 (SIEMENS)
   RUNG wire#powerrail
      Contact( "LBP_Chan7".MDyn[44] )
      I_Contact( "DB365_M_UNIT_02_STA_4".M_CODES_UNIT_02_STA_4.Ack_M44 )
      I_Contact( "DB2120_MPP_ITC_IPC".RESET_FAULTS )
      I_Contact( "DB365_M_UNIT_02_STA_4".M_CODES_UNIT_02_STA_4.M_RESET_PULSE )
      Coil( "DB365_M_UNIT_02_STA_4".M_CODES_UNIT_02_STA_4.M44 )
   END_RUNG
   // the same network as SCL:
   "DB365_M_UNIT_02_STA_4".M_CODES_UNIT_02_STA_4.M44 := "LBP_Chan7".MDyn[44] AND NOT "DB365_M_UNIT_02_STA_4".M_CODES_UNIT_02_STA_4.Ack_M44 AND NOT "DB2120_MPP_ITC_IPC".RESET_FAULTS AND NOT "DB365_M_UNIT_02_STA_4".M_CODES_UNIT_02_STA_4.M_RESET_PULSE;
END_REGION

REGION Network 43: ACKNOWLEDGE M45-GEAR STAGE 5 (SIEMENS) / ACKNOWLEDGE M45-SHIFT REDUCTION 5 (SIEMENS)
   RUNG wire#powerrail
      Contact( "M_ZERO" )
      Coil( "DB365_M_UNIT_02_STA_4".M_CODES_UNIT_02_STA_4.Ack_M45 )
   END_RUNG
   // the same network as SCL:
   "DB365_M_UNIT_02_STA_4".M_CODES_UNIT_02_STA_4.Ack_M45 := "M_ZERO";
END_REGION

REGION Network 44: M45-GEAR STAGE 5 (SIEMENS) / M45-SHIFT REDUCTION 5 (SIEMENS)
   RUNG wire#powerrail
      Contact( "LBP_Chan7".MDyn[45] )
      I_Contact( "DB365_M_UNIT_02_STA_4".M_CODES_UNIT_02_STA_4.Ack_M45 )
      I_Contact( "DB2120_MPP_ITC_IPC".RESET_FAULTS )
      I_Contact( "DB365_M_UNIT_02_STA_4".M_CODES_UNIT_02_STA_4.M_RESET_PULSE )
      Coil( "DB365_M_UNIT_02_STA_4".M_CODES_UNIT_02_STA_4.M45 )
   END_RUNG
   // the same network as SCL:
   "DB365_M_UNIT_02_STA_4".M_CODES_UNIT_02_STA_4.M45 := "LBP_Chan7".MDyn[45] AND NOT "DB365_M_UNIT_02_STA_4".M_CODES_UNIT_02_STA_4.Ack_M45 AND NOT "DB2120_MPP_ITC_IPC".RESET_FAULTS AND NOT "DB365_M_UNIT_02_STA_4".M_CODES_UNIT_02_STA_4.M_RESET_PULSE;
END_REGION

REGION Network 45: ACKNOWLEDGE M70-SPINDLE IS SWITCHED TO AXIS MODE (SIEMENS) / ACKNOWLEDGE M42-SHIFT REDUCTION 2 (SIEMENS)
   RUNG wire#powerrail
      Contact( "M_ZERO" )
      Coil( "DB365_M_UNIT_02_STA_4".M_CODES_UNIT_02_STA_4.Ack_M70 )
   END_RUNG
   // the same network as SCL:
   "DB365_M_UNIT_02_STA_4".M_CODES_UNIT_02_STA_4.Ack_M70 := "M_ZERO";
END_REGION

REGION Network 46: M70-SPINDLE IS SWITCHED TO AXIS MODE (SIEMENS) / M42-SHIFT REDUCTION 2 (SIEMENS)
   RUNG wire#powerrail
      Contact( "LBP_Chan7".MDyn[70] )
      I_Contact( "DB365_M_UNIT_02_STA_4".M_CODES_UNIT_02_STA_4.Ack_M70 )
      I_Contact( "DB2120_MPP_ITC_IPC".RESET_FAULTS )
      I_Contact( "DB365_M_UNIT_02_STA_4".M_CODES_UNIT_02_STA_4.M_RESET_PULSE )
      Coil( "DB365_M_UNIT_02_STA_4".M_CODES_UNIT_02_STA_4.M70 )
   END_RUNG
   // the same network as SCL:
   "DB365_M_UNIT_02_STA_4".M_CODES_UNIT_02_STA_4.M70 := "LBP_Chan7".MDyn[70] AND NOT "DB365_M_UNIT_02_STA_4".M_CODES_UNIT_02_STA_4.Ack_M70 AND NOT "DB2120_MPP_ITC_IPC".RESET_FAULTS AND NOT "DB365_M_UNIT_02_STA_4".M_CODES_UNIT_02_STA_4.M_RESET_PULSE;
END_REGION

REGION Network 47: ACKNOWLEDGE M98-EXTERNAL LANGUAGE (SIEMENS) / ACKNOWLEDGE M42-SHIFT REDUCTION 2 (SIEMENS)
   RUNG wire#powerrail
      Contact( "M_ZERO" )
      Coil( "DB365_M_UNIT_02_STA_4".M_CODES_UNIT_02_STA_4.Ack_M98 )
   END_RUNG
   // the same network as SCL:
   "DB365_M_UNIT_02_STA_4".M_CODES_UNIT_02_STA_4.Ack_M98 := "M_ZERO";
END_REGION

REGION Network 48: M98-EXTERNAL LANGUAGE (SIEMENS) / M42-SHIFT REDUCTION 2 (SIEMENS)
   RUNG wire#powerrail
      Contact( "LBP_Chan7".MDyn[98] )
      I_Contact( "DB365_M_UNIT_02_STA_4".M_CODES_UNIT_02_STA_4.Ack_M98 )
      I_Contact( "DB2120_MPP_ITC_IPC".RESET_FAULTS )
      I_Contact( "DB365_M_UNIT_02_STA_4".M_CODES_UNIT_02_STA_4.M_RESET_PULSE )
      Coil( "DB365_M_UNIT_02_STA_4".M_CODES_UNIT_02_STA_4.M98 )
   END_RUNG
   // the same network as SCL:
   "DB365_M_UNIT_02_STA_4".M_CODES_UNIT_02_STA_4.M98 := "LBP_Chan7".MDyn[98] AND NOT "DB365_M_UNIT_02_STA_4".M_CODES_UNIT_02_STA_4.Ack_M98 AND NOT "DB2120_MPP_ITC_IPC".RESET_FAULTS AND NOT "DB365_M_UNIT_02_STA_4".M_CODES_UNIT_02_STA_4.M_RESET_PULSE;
END_REGION

REGION Network 49: ACKNOWLEDGE M99-EXTERNAL LANGUAGE (SIEMENS) / ACKNOWLEDGE M42-SHIFT REDUCTION 2 (SIEMENS)
   RUNG wire#powerrail
      Contact( "M_ZERO" )
      Coil( "DB365_M_UNIT_02_STA_4".M_CODES_UNIT_02_STA_4.Ack_M99 )
   END_RUNG
   // the same network as SCL:
   "DB365_M_UNIT_02_STA_4".M_CODES_UNIT_02_STA_4.Ack_M99 := "M_ZERO";
END_REGION

REGION Network 50: M99-EXTERNAL LANGUAGE (SIEMENS) / M42-SHIFT REDUCTION 2 (SIEMENS)
   RUNG wire#powerrail
      Contact( "LBP_Chan7".MDyn[99] )
      I_Contact( "DB365_M_UNIT_02_STA_4".M_CODES_UNIT_02_STA_4.Ack_M99 )
      I_Contact( "DB2120_MPP_ITC_IPC".RESET_FAULTS )
      I_Contact( "DB365_M_UNIT_02_STA_4".M_CODES_UNIT_02_STA_4.M_RESET_PULSE )
      Coil( "DB365_M_UNIT_02_STA_4".M_CODES_UNIT_02_STA_4.M99 )
   END_RUNG
   // the same network as SCL:
   "DB365_M_UNIT_02_STA_4".M_CODES_UNIT_02_STA_4.M99 := "LBP_Chan7".MDyn[99] AND NOT "DB365_M_UNIT_02_STA_4".M_CODES_UNIT_02_STA_4.Ack_M99 AND NOT "DB2120_MPP_ITC_IPC".RESET_FAULTS AND NOT "DB365_M_UNIT_02_STA_4".M_CODES_UNIT_02_STA_4.M_RESET_PULSE;
END_REGION

REGION Network 51: ACKNOWLEDGE M100-WAIT UNTIL E10 IN POSITION FIXTURE 1 STATION 1(READ-IN DISABLE) / ACKNOWLEDGE M23-SWITCH ON SPINDLE FRAME BLOWING
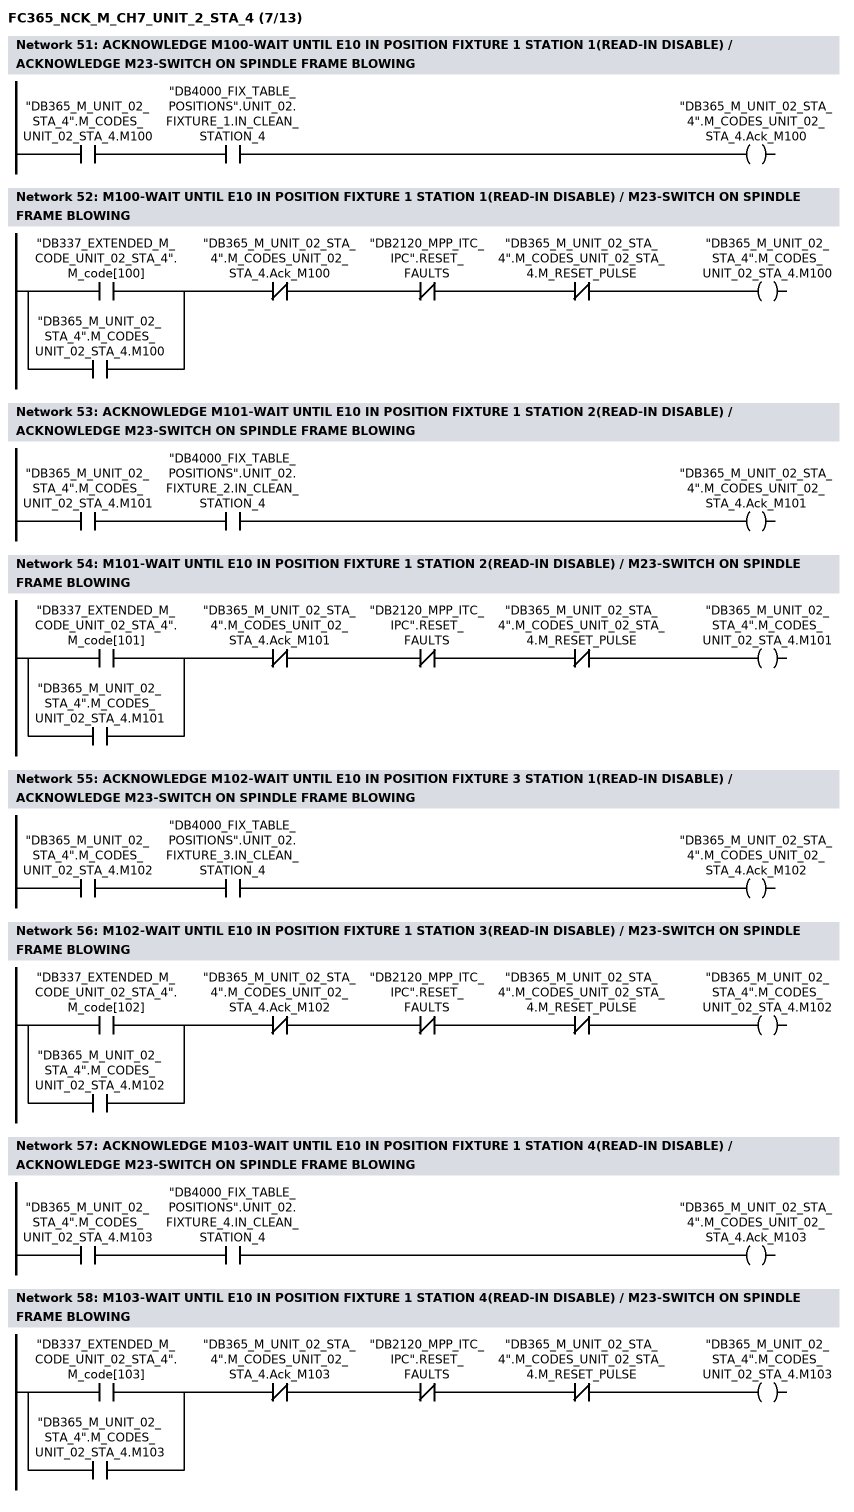
   RUNG wire#powerrail
      Contact( "DB365_M_UNIT_02_STA_4".M_CODES_UNIT_02_STA_4.M100 )
      Contact( "DB4000_FIX_TABLE_POSITIONS".UNIT_02.FIXTURE_1.IN_CLEAN_STATION_4 )
      Coil( "DB365_M_UNIT_02_STA_4".M_CODES_UNIT_02_STA_4.Ack_M100 )
   END_RUNG
   // the same network as SCL:
   "DB365_M_UNIT_02_STA_4".M_CODES_UNIT_02_STA_4.Ack_M100 := "DB365_M_UNIT_02_STA_4".M_CODES_UNIT_02_STA_4.M100 AND "DB4000_FIX_TABLE_POSITIONS".UNIT_02.FIXTURE_1.IN_CLEAN_STATION_4;
END_REGION

REGION Network 52: M100-WAIT UNTIL E10 IN POSITION FIXTURE 1 STATION 1(READ-IN DISABLE) / M23-SWITCH ON SPINDLE FRAME BLOWING
   RUNG wire#powerrail
      Contact( "DB337_EXTENDED_M_CODE_UNIT_02_STA_4".M_code[100] )
      wire#w1
      I_Contact( "DB365_M_UNIT_02_STA_4".M_CODES_UNIT_02_STA_4.Ack_M100 )
      I_Contact( "DB2120_MPP_ITC_IPC".RESET_FAULTS )
      I_Contact( "DB365_M_UNIT_02_STA_4".M_CODES_UNIT_02_STA_4.M_RESET_PULSE )
      Coil( "DB365_M_UNIT_02_STA_4".M_CODES_UNIT_02_STA_4.M100 )
   END_RUNG
   RUNG wire#powerrail
      Contact( "DB365_M_UNIT_02_STA_4".M_CODES_UNIT_02_STA_4.M100 )
   END_RUNG wire#w1
   // the same network as SCL:
   "DB365_M_UNIT_02_STA_4".M_CODES_UNIT_02_STA_4.M100 := ("DB337_EXTENDED_M_CODE_UNIT_02_STA_4".M_code[100] OR "DB365_M_UNIT_02_STA_4".M_CODES_UNIT_02_STA_4.M100) AND NOT "DB365_M_UNIT_02_STA_4".M_CODES_UNIT_02_STA_4.Ack_M100 AND NOT "DB2120_MPP_ITC_IPC".RESET_FAULTS AND NOT "DB365_M_UNIT_02_STA_4".M_CODES_UNIT_02_STA_4.M_RESET_PULSE;
END_REGION

REGION Network 53: ACKNOWLEDGE M101-WAIT UNTIL E10 IN POSITION FIXTURE 1 STATION 2(READ-IN DISABLE) / ACKNOWLEDGE M23-SWITCH ON SPINDLE FRAME BLOWING
   RUNG wire#powerrail
      Contact( "DB365_M_UNIT_02_STA_4".M_CODES_UNIT_02_STA_4.M101 )
      Contact( "DB4000_FIX_TABLE_POSITIONS".UNIT_02.FIXTURE_2.IN_CLEAN_STATION_4 )
      Coil( "DB365_M_UNIT_02_STA_4".M_CODES_UNIT_02_STA_4.Ack_M101 )
   END_RUNG
   // the same network as SCL:
   "DB365_M_UNIT_02_STA_4".M_CODES_UNIT_02_STA_4.Ack_M101 := "DB365_M_UNIT_02_STA_4".M_CODES_UNIT_02_STA_4.M101 AND "DB4000_FIX_TABLE_POSITIONS".UNIT_02.FIXTURE_2.IN_CLEAN_STATION_4;
END_REGION

REGION Network 54: M101-WAIT UNTIL E10 IN POSITION FIXTURE 1 STATION 2(READ-IN DISABLE) / M23-SWITCH ON SPINDLE FRAME BLOWING
   RUNG wire#powerrail
      Contact( "DB337_EXTENDED_M_CODE_UNIT_02_STA_4".M_code[101] )
      wire#w1
      I_Contact( "DB365_M_UNIT_02_STA_4".M_CODES_UNIT_02_STA_4.Ack_M101 )
      I_Contact( "DB2120_MPP_ITC_IPC".RESET_FAULTS )
      I_Contact( "DB365_M_UNIT_02_STA_4".M_CODES_UNIT_02_STA_4.M_RESET_PULSE )
      Coil( "DB365_M_UNIT_02_STA_4".M_CODES_UNIT_02_STA_4.M101 )
   END_RUNG
   RUNG wire#powerrail
      Contact( "DB365_M_UNIT_02_STA_4".M_CODES_UNIT_02_STA_4.M101 )
   END_RUNG wire#w1
   // the same network as SCL:
   "DB365_M_UNIT_02_STA_4".M_CODES_UNIT_02_STA_4.M101 := ("DB337_EXTENDED_M_CODE_UNIT_02_STA_4".M_code[101] OR "DB365_M_UNIT_02_STA_4".M_CODES_UNIT_02_STA_4.M101) AND NOT "DB365_M_UNIT_02_STA_4".M_CODES_UNIT_02_STA_4.Ack_M101 AND NOT "DB2120_MPP_ITC_IPC".RESET_FAULTS AND NOT "DB365_M_UNIT_02_STA_4".M_CODES_UNIT_02_STA_4.M_RESET_PULSE;
END_REGION

REGION Network 55: ACKNOWLEDGE M102-WAIT UNTIL E10 IN POSITION FIXTURE 3 STATION 1(READ-IN DISABLE) / ACKNOWLEDGE M23-SWITCH ON SPINDLE FRAME BLOWING
   RUNG wire#powerrail
      Contact( "DB365_M_UNIT_02_STA_4".M_CODES_UNIT_02_STA_4.M102 )
      Contact( "DB4000_FIX_TABLE_POSITIONS".UNIT_02.FIXTURE_3.IN_CLEAN_STATION_4 )
      Coil( "DB365_M_UNIT_02_STA_4".M_CODES_UNIT_02_STA_4.Ack_M102 )
   END_RUNG
   // the same network as SCL:
   "DB365_M_UNIT_02_STA_4".M_CODES_UNIT_02_STA_4.Ack_M102 := "DB365_M_UNIT_02_STA_4".M_CODES_UNIT_02_STA_4.M102 AND "DB4000_FIX_TABLE_POSITIONS".UNIT_02.FIXTURE_3.IN_CLEAN_STATION_4;
END_REGION

REGION Network 56: M102-WAIT UNTIL E10 IN POSITION FIXTURE 1 STATION 3(READ-IN DISABLE) / M23-SWITCH ON SPINDLE FRAME BLOWING
   RUNG wire#powerrail
      Contact( "DB337_EXTENDED_M_CODE_UNIT_02_STA_4".M_code[102] )
      wire#w1
      I_Contact( "DB365_M_UNIT_02_STA_4".M_CODES_UNIT_02_STA_4.Ack_M102 )
      I_Contact( "DB2120_MPP_ITC_IPC".RESET_FAULTS )
      I_Contact( "DB365_M_UNIT_02_STA_4".M_CODES_UNIT_02_STA_4.M_RESET_PULSE )
      Coil( "DB365_M_UNIT_02_STA_4".M_CODES_UNIT_02_STA_4.M102 )
   END_RUNG
   RUNG wire#powerrail
      Contact( "DB365_M_UNIT_02_STA_4".M_CODES_UNIT_02_STA_4.M102 )
   END_RUNG wire#w1
   // the same network as SCL:
   "DB365_M_UNIT_02_STA_4".M_CODES_UNIT_02_STA_4.M102 := ("DB337_EXTENDED_M_CODE_UNIT_02_STA_4".M_code[102] OR "DB365_M_UNIT_02_STA_4".M_CODES_UNIT_02_STA_4.M102) AND NOT "DB365_M_UNIT_02_STA_4".M_CODES_UNIT_02_STA_4.Ack_M102 AND NOT "DB2120_MPP_ITC_IPC".RESET_FAULTS AND NOT "DB365_M_UNIT_02_STA_4".M_CODES_UNIT_02_STA_4.M_RESET_PULSE;
END_REGION

REGION Network 57: ACKNOWLEDGE M103-WAIT UNTIL E10 IN POSITION FIXTURE 1 STATION 4(READ-IN DISABLE) / ACKNOWLEDGE M23-SWITCH ON SPINDLE FRAME BLOWING
   RUNG wire#powerrail
      Contact( "DB365_M_UNIT_02_STA_4".M_CODES_UNIT_02_STA_4.M103 )
      Contact( "DB4000_FIX_TABLE_POSITIONS".UNIT_02.FIXTURE_4.IN_CLEAN_STATION_4 )
      Coil( "DB365_M_UNIT_02_STA_4".M_CODES_UNIT_02_STA_4.Ack_M103 )
   END_RUNG
   // the same network as SCL:
   "DB365_M_UNIT_02_STA_4".M_CODES_UNIT_02_STA_4.Ack_M103 := "DB365_M_UNIT_02_STA_4".M_CODES_UNIT_02_STA_4.M103 AND "DB4000_FIX_TABLE_POSITIONS".UNIT_02.FIXTURE_4.IN_CLEAN_STATION_4;
END_REGION

REGION Network 58: M103-WAIT UNTIL E10 IN POSITION FIXTURE 1 STATION 4(READ-IN DISABLE) / M23-SWITCH ON SPINDLE FRAME BLOWING
   RUNG wire#powerrail
      Contact( "DB337_EXTENDED_M_CODE_UNIT_02_STA_4".M_code[103] )
      wire#w1
      I_Contact( "DB365_M_UNIT_02_STA_4".M_CODES_UNIT_02_STA_4.Ack_M103 )
      I_Contact( "DB2120_MPP_ITC_IPC".RESET_FAULTS )
      I_Contact( "DB365_M_UNIT_02_STA_4".M_CODES_UNIT_02_STA_4.M_RESET_PULSE )
      Coil( "DB365_M_UNIT_02_STA_4".M_CODES_UNIT_02_STA_4.M103 )
   END_RUNG
   RUNG wire#powerrail
      Contact( "DB365_M_UNIT_02_STA_4".M_CODES_UNIT_02_STA_4.M103 )
   END_RUNG wire#w1
   // the same network as SCL:
   "DB365_M_UNIT_02_STA_4".M_CODES_UNIT_02_STA_4.M103 := ("DB337_EXTENDED_M_CODE_UNIT_02_STA_4".M_code[103] OR "DB365_M_UNIT_02_STA_4".M_CODES_UNIT_02_STA_4.M103) AND NOT "DB365_M_UNIT_02_STA_4".M_CODES_UNIT_02_STA_4.Ack_M103 AND NOT "DB2120_MPP_ITC_IPC".RESET_FAULTS AND NOT "DB365_M_UNIT_02_STA_4".M_CODES_UNIT_02_STA_4.M_RESET_PULSE;
END_REGION

REGION Network 59: ACKNOWLEDGE M110-UNBLOCK TABLE
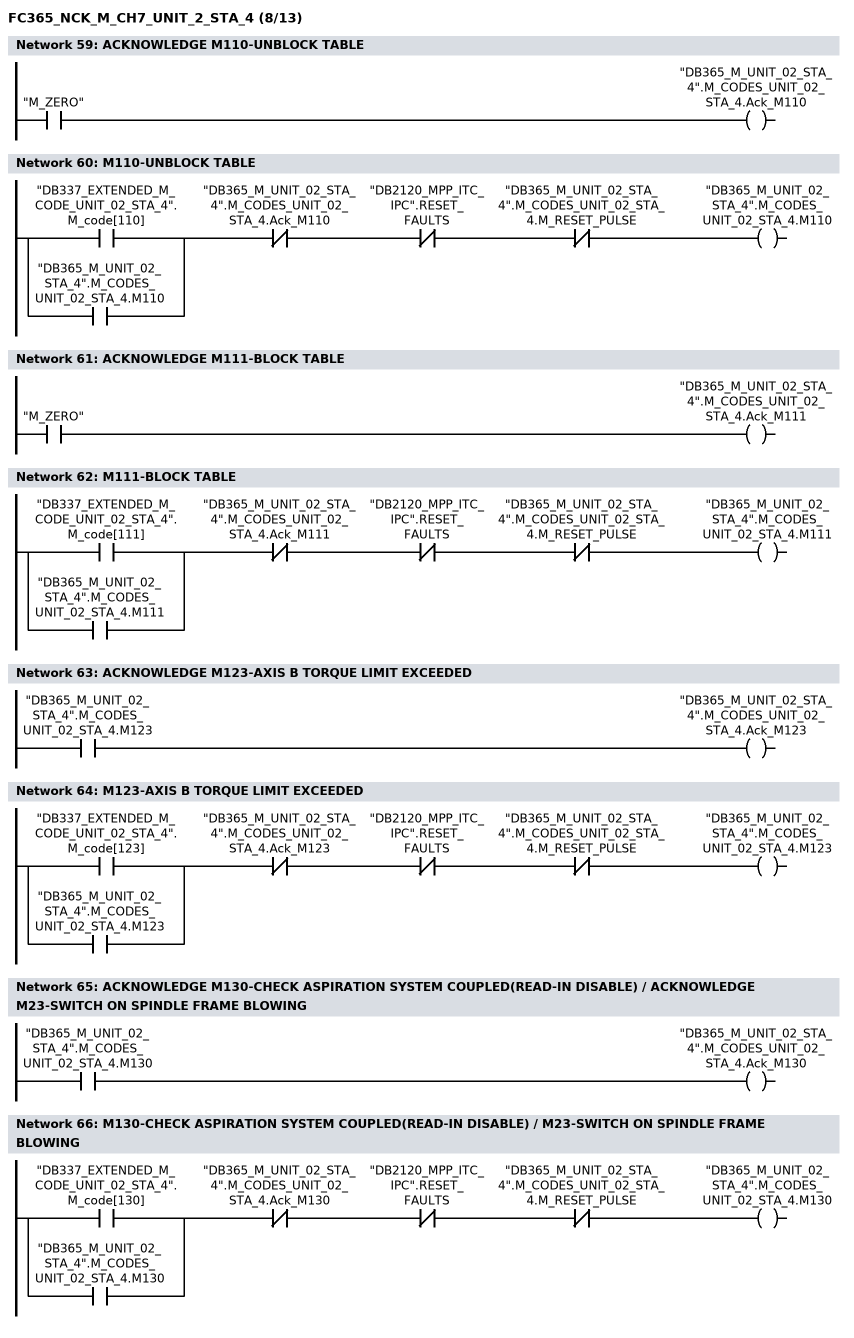
   RUNG wire#powerrail
      Contact( "M_ZERO" )
      Coil( "DB365_M_UNIT_02_STA_4".M_CODES_UNIT_02_STA_4.Ack_M110 )
   END_RUNG
   // the same network as SCL:
   "DB365_M_UNIT_02_STA_4".M_CODES_UNIT_02_STA_4.Ack_M110 := "M_ZERO";
END_REGION

REGION Network 60: M110-UNBLOCK TABLE
   RUNG wire#powerrail
      Contact( "DB337_EXTENDED_M_CODE_UNIT_02_STA_4".M_code[110] )
      wire#w1
      I_Contact( "DB365_M_UNIT_02_STA_4".M_CODES_UNIT_02_STA_4.Ack_M110 )
      I_Contact( "DB2120_MPP_ITC_IPC".RESET_FAULTS )
      I_Contact( "DB365_M_UNIT_02_STA_4".M_CODES_UNIT_02_STA_4.M_RESET_PULSE )
      Coil( "DB365_M_UNIT_02_STA_4".M_CODES_UNIT_02_STA_4.M110 )
   END_RUNG
   RUNG wire#powerrail
      Contact( "DB365_M_UNIT_02_STA_4".M_CODES_UNIT_02_STA_4.M110 )
   END_RUNG wire#w1
   // the same network as SCL:
   "DB365_M_UNIT_02_STA_4".M_CODES_UNIT_02_STA_4.M110 := ("DB337_EXTENDED_M_CODE_UNIT_02_STA_4".M_code[110] OR "DB365_M_UNIT_02_STA_4".M_CODES_UNIT_02_STA_4.M110) AND NOT "DB365_M_UNIT_02_STA_4".M_CODES_UNIT_02_STA_4.Ack_M110 AND NOT "DB2120_MPP_ITC_IPC".RESET_FAULTS AND NOT "DB365_M_UNIT_02_STA_4".M_CODES_UNIT_02_STA_4.M_RESET_PULSE;
END_REGION

REGION Network 61: ACKNOWLEDGE M111-BLOCK TABLE
   RUNG wire#powerrail
      Contact( "M_ZERO" )
      Coil( "DB365_M_UNIT_02_STA_4".M_CODES_UNIT_02_STA_4.Ack_M111 )
   END_RUNG
   // the same network as SCL:
   "DB365_M_UNIT_02_STA_4".M_CODES_UNIT_02_STA_4.Ack_M111 := "M_ZERO";
END_REGION

REGION Network 62: M111-BLOCK TABLE
   RUNG wire#powerrail
      Contact( "DB337_EXTENDED_M_CODE_UNIT_02_STA_4".M_code[111] )
      wire#w1
      I_Contact( "DB365_M_UNIT_02_STA_4".M_CODES_UNIT_02_STA_4.Ack_M111 )
      I_Contact( "DB2120_MPP_ITC_IPC".RESET_FAULTS )
      I_Contact( "DB365_M_UNIT_02_STA_4".M_CODES_UNIT_02_STA_4.M_RESET_PULSE )
      Coil( "DB365_M_UNIT_02_STA_4".M_CODES_UNIT_02_STA_4.M111 )
   END_RUNG
   RUNG wire#powerrail
      Contact( "DB365_M_UNIT_02_STA_4".M_CODES_UNIT_02_STA_4.M111 )
   END_RUNG wire#w1
   // the same network as SCL:
   "DB365_M_UNIT_02_STA_4".M_CODES_UNIT_02_STA_4.M111 := ("DB337_EXTENDED_M_CODE_UNIT_02_STA_4".M_code[111] OR "DB365_M_UNIT_02_STA_4".M_CODES_UNIT_02_STA_4.M111) AND NOT "DB365_M_UNIT_02_STA_4".M_CODES_UNIT_02_STA_4.Ack_M111 AND NOT "DB2120_MPP_ITC_IPC".RESET_FAULTS AND NOT "DB365_M_UNIT_02_STA_4".M_CODES_UNIT_02_STA_4.M_RESET_PULSE;
END_REGION

REGION Network 63: ACKNOWLEDGE M123-AXIS B TORQUE LIMIT EXCEEDED
   RUNG wire#powerrail
      Contact( "DB365_M_UNIT_02_STA_4".M_CODES_UNIT_02_STA_4.M123 )
      Coil( "DB365_M_UNIT_02_STA_4".M_CODES_UNIT_02_STA_4.Ack_M123 )
   END_RUNG
   // the same network as SCL:
   "DB365_M_UNIT_02_STA_4".M_CODES_UNIT_02_STA_4.Ack_M123 := "DB365_M_UNIT_02_STA_4".M_CODES_UNIT_02_STA_4.M123;
END_REGION

REGION Network 64: M123-AXIS B TORQUE LIMIT EXCEEDED
   RUNG wire#powerrail
      Contact( "DB337_EXTENDED_M_CODE_UNIT_02_STA_4".M_code[123] )
      wire#w1
      I_Contact( "DB365_M_UNIT_02_STA_4".M_CODES_UNIT_02_STA_4.Ack_M123 )
      I_Contact( "DB2120_MPP_ITC_IPC".RESET_FAULTS )
      I_Contact( "DB365_M_UNIT_02_STA_4".M_CODES_UNIT_02_STA_4.M_RESET_PULSE )
      Coil( "DB365_M_UNIT_02_STA_4".M_CODES_UNIT_02_STA_4.M123 )
   END_RUNG
   RUNG wire#powerrail
      Contact( "DB365_M_UNIT_02_STA_4".M_CODES_UNIT_02_STA_4.M123 )
   END_RUNG wire#w1
   // the same network as SCL:
   "DB365_M_UNIT_02_STA_4".M_CODES_UNIT_02_STA_4.M123 := ("DB337_EXTENDED_M_CODE_UNIT_02_STA_4".M_code[123] OR "DB365_M_UNIT_02_STA_4".M_CODES_UNIT_02_STA_4.M123) AND NOT "DB365_M_UNIT_02_STA_4".M_CODES_UNIT_02_STA_4.Ack_M123 AND NOT "DB2120_MPP_ITC_IPC".RESET_FAULTS AND NOT "DB365_M_UNIT_02_STA_4".M_CODES_UNIT_02_STA_4.M_RESET_PULSE;
END_REGION

REGION Network 65: ACKNOWLEDGE M130-CHECK ASPIRATION SYSTEM COUPLED(READ-IN DISABLE) / ACKNOWLEDGE M23-SWITCH ON SPINDLE FRAME BLOWING
   RUNG wire#powerrail
      Contact( "DB365_M_UNIT_02_STA_4".M_CODES_UNIT_02_STA_4.M130 )
      Coil( "DB365_M_UNIT_02_STA_4".M_CODES_UNIT_02_STA_4.Ack_M130 )
   END_RUNG
   // the same network as SCL:
   "DB365_M_UNIT_02_STA_4".M_CODES_UNIT_02_STA_4.Ack_M130 := "DB365_M_UNIT_02_STA_4".M_CODES_UNIT_02_STA_4.M130;
END_REGION

REGION Network 66: M130-CHECK ASPIRATION SYSTEM COUPLED(READ-IN DISABLE) / M23-SWITCH ON SPINDLE FRAME BLOWING
   RUNG wire#powerrail
      Contact( "DB337_EXTENDED_M_CODE_UNIT_02_STA_4".M_code[130] )
      wire#w1
      I_Contact( "DB365_M_UNIT_02_STA_4".M_CODES_UNIT_02_STA_4.Ack_M130 )
      I_Contact( "DB2120_MPP_ITC_IPC".RESET_FAULTS )
      I_Contact( "DB365_M_UNIT_02_STA_4".M_CODES_UNIT_02_STA_4.M_RESET_PULSE )
      Coil( "DB365_M_UNIT_02_STA_4".M_CODES_UNIT_02_STA_4.M130 )
   END_RUNG
   RUNG wire#powerrail
      Contact( "DB365_M_UNIT_02_STA_4".M_CODES_UNIT_02_STA_4.M130 )
   END_RUNG wire#w1
   // the same network as SCL:
   "DB365_M_UNIT_02_STA_4".M_CODES_UNIT_02_STA_4.M130 := ("DB337_EXTENDED_M_CODE_UNIT_02_STA_4".M_code[130] OR "DB365_M_UNIT_02_STA_4".M_CODES_UNIT_02_STA_4.M130) AND NOT "DB365_M_UNIT_02_STA_4".M_CODES_UNIT_02_STA_4.Ack_M130 AND NOT "DB2120_MPP_ITC_IPC".RESET_FAULTS AND NOT "DB365_M_UNIT_02_STA_4".M_CODES_UNIT_02_STA_4.M_RESET_PULSE;
END_REGION

REGION Network 67: ACKNOWLEDGE M131-CHECK ASPIRATION SYSTEM UNCOUPLED(READ-IN DISABLE) / ACKNOWLEDGE M23-SWITCH ON SPINDLE FRAME BLOWING
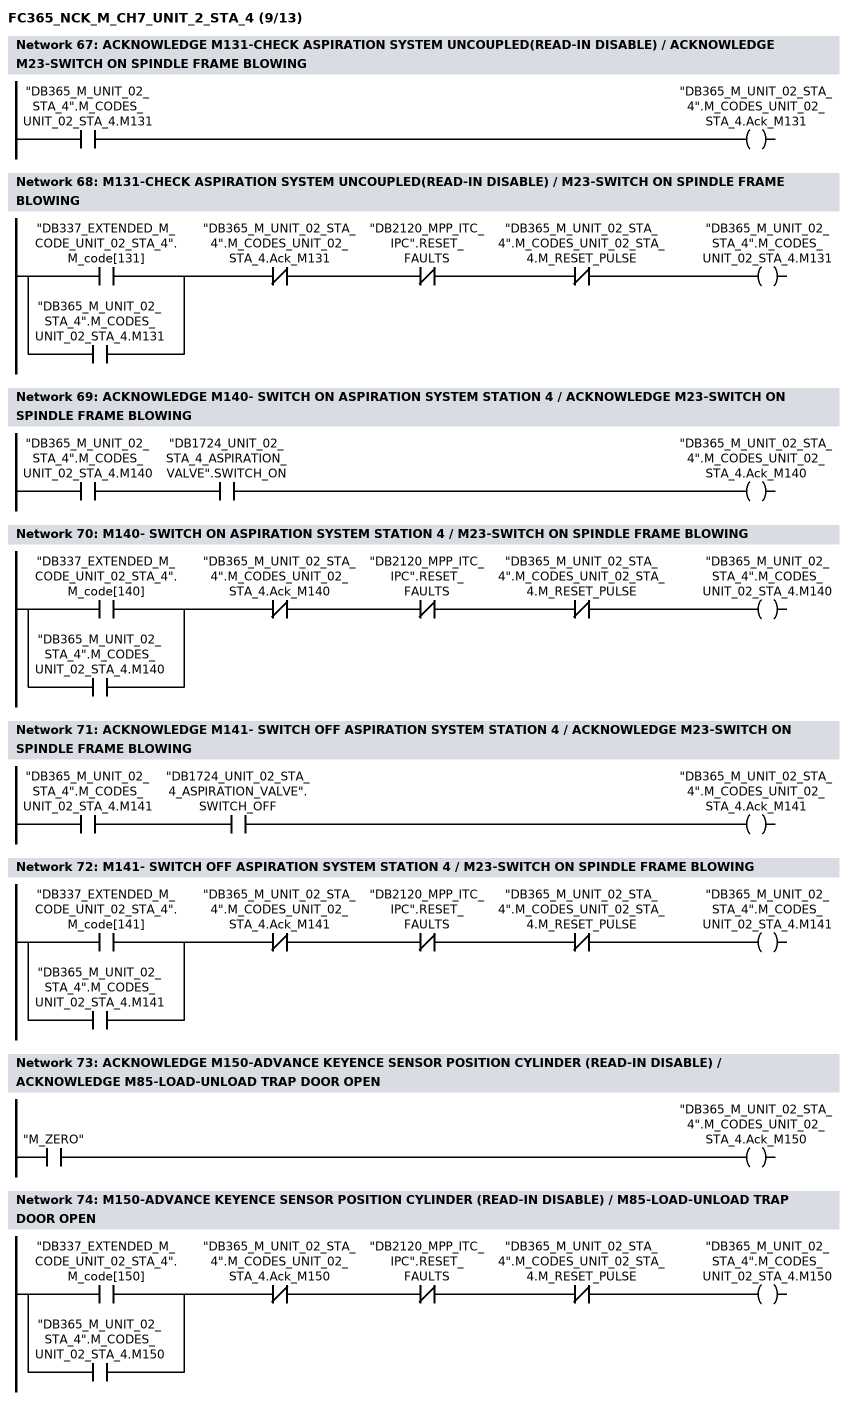
   RUNG wire#powerrail
      Contact( "DB365_M_UNIT_02_STA_4".M_CODES_UNIT_02_STA_4.M131 )
      Coil( "DB365_M_UNIT_02_STA_4".M_CODES_UNIT_02_STA_4.Ack_M131 )
   END_RUNG
   // the same network as SCL:
   "DB365_M_UNIT_02_STA_4".M_CODES_UNIT_02_STA_4.Ack_M131 := "DB365_M_UNIT_02_STA_4".M_CODES_UNIT_02_STA_4.M131;
END_REGION

REGION Network 68: M131-CHECK ASPIRATION SYSTEM UNCOUPLED(READ-IN DISABLE) / M23-SWITCH ON SPINDLE FRAME BLOWING
   RUNG wire#powerrail
      Contact( "DB337_EXTENDED_M_CODE_UNIT_02_STA_4".M_code[131] )
      wire#w1
      I_Contact( "DB365_M_UNIT_02_STA_4".M_CODES_UNIT_02_STA_4.Ack_M131 )
      I_Contact( "DB2120_MPP_ITC_IPC".RESET_FAULTS )
      I_Contact( "DB365_M_UNIT_02_STA_4".M_CODES_UNIT_02_STA_4.M_RESET_PULSE )
      Coil( "DB365_M_UNIT_02_STA_4".M_CODES_UNIT_02_STA_4.M131 )
   END_RUNG
   RUNG wire#powerrail
      Contact( "DB365_M_UNIT_02_STA_4".M_CODES_UNIT_02_STA_4.M131 )
   END_RUNG wire#w1
   // the same network as SCL:
   "DB365_M_UNIT_02_STA_4".M_CODES_UNIT_02_STA_4.M131 := ("DB337_EXTENDED_M_CODE_UNIT_02_STA_4".M_code[131] OR "DB365_M_UNIT_02_STA_4".M_CODES_UNIT_02_STA_4.M131) AND NOT "DB365_M_UNIT_02_STA_4".M_CODES_UNIT_02_STA_4.Ack_M131 AND NOT "DB2120_MPP_ITC_IPC".RESET_FAULTS AND NOT "DB365_M_UNIT_02_STA_4".M_CODES_UNIT_02_STA_4.M_RESET_PULSE;
END_REGION

REGION Network 69: ACKNOWLEDGE M140- SWITCH ON ASPIRATION SYSTEM STATION 4 / ACKNOWLEDGE M23-SWITCH ON SPINDLE FRAME BLOWING
   RUNG wire#powerrail
      Contact( "DB365_M_UNIT_02_STA_4".M_CODES_UNIT_02_STA_4.M140 )
      Contact( "DB1724_UNIT_02_STA_4_ASPIRATION_VALVE".SWITCH_ON )
      Coil( "DB365_M_UNIT_02_STA_4".M_CODES_UNIT_02_STA_4.Ack_M140 )
   END_RUNG
   // the same network as SCL:
   "DB365_M_UNIT_02_STA_4".M_CODES_UNIT_02_STA_4.Ack_M140 := "DB365_M_UNIT_02_STA_4".M_CODES_UNIT_02_STA_4.M140 AND "DB1724_UNIT_02_STA_4_ASPIRATION_VALVE".SWITCH_ON;
END_REGION

REGION Network 70: M140- SWITCH ON ASPIRATION SYSTEM STATION 4 / M23-SWITCH ON SPINDLE FRAME BLOWING
   RUNG wire#powerrail
      Contact( "DB337_EXTENDED_M_CODE_UNIT_02_STA_4".M_code[140] )
      wire#w1
      I_Contact( "DB365_M_UNIT_02_STA_4".M_CODES_UNIT_02_STA_4.Ack_M140 )
      I_Contact( "DB2120_MPP_ITC_IPC".RESET_FAULTS )
      I_Contact( "DB365_M_UNIT_02_STA_4".M_CODES_UNIT_02_STA_4.M_RESET_PULSE )
      Coil( "DB365_M_UNIT_02_STA_4".M_CODES_UNIT_02_STA_4.M140 )
   END_RUNG
   RUNG wire#powerrail
      Contact( "DB365_M_UNIT_02_STA_4".M_CODES_UNIT_02_STA_4.M140 )
   END_RUNG wire#w1
   // the same network as SCL:
   "DB365_M_UNIT_02_STA_4".M_CODES_UNIT_02_STA_4.M140 := ("DB337_EXTENDED_M_CODE_UNIT_02_STA_4".M_code[140] OR "DB365_M_UNIT_02_STA_4".M_CODES_UNIT_02_STA_4.M140) AND NOT "DB365_M_UNIT_02_STA_4".M_CODES_UNIT_02_STA_4.Ack_M140 AND NOT "DB2120_MPP_ITC_IPC".RESET_FAULTS AND NOT "DB365_M_UNIT_02_STA_4".M_CODES_UNIT_02_STA_4.M_RESET_PULSE;
END_REGION

REGION Network 71: ACKNOWLEDGE M141- SWITCH OFF ASPIRATION SYSTEM STATION 4 / ACKNOWLEDGE M23-SWITCH ON SPINDLE FRAME BLOWING
   RUNG wire#powerrail
      Contact( "DB365_M_UNIT_02_STA_4".M_CODES_UNIT_02_STA_4.M141 )
      Contact( "DB1724_UNIT_02_STA_4_ASPIRATION_VALVE".SWITCH_OFF )
      Coil( "DB365_M_UNIT_02_STA_4".M_CODES_UNIT_02_STA_4.Ack_M141 )
   END_RUNG
   // the same network as SCL:
   "DB365_M_UNIT_02_STA_4".M_CODES_UNIT_02_STA_4.Ack_M141 := "DB365_M_UNIT_02_STA_4".M_CODES_UNIT_02_STA_4.M141 AND "DB1724_UNIT_02_STA_4_ASPIRATION_VALVE".SWITCH_OFF;
END_REGION

REGION Network 72: M141- SWITCH OFF ASPIRATION SYSTEM STATION 4 / M23-SWITCH ON SPINDLE FRAME BLOWING
   RUNG wire#powerrail
      Contact( "DB337_EXTENDED_M_CODE_UNIT_02_STA_4".M_code[141] )
      wire#w1
      I_Contact( "DB365_M_UNIT_02_STA_4".M_CODES_UNIT_02_STA_4.Ack_M141 )
      I_Contact( "DB2120_MPP_ITC_IPC".RESET_FAULTS )
      I_Contact( "DB365_M_UNIT_02_STA_4".M_CODES_UNIT_02_STA_4.M_RESET_PULSE )
      Coil( "DB365_M_UNIT_02_STA_4".M_CODES_UNIT_02_STA_4.M141 )
   END_RUNG
   RUNG wire#powerrail
      Contact( "DB365_M_UNIT_02_STA_4".M_CODES_UNIT_02_STA_4.M141 )
   END_RUNG wire#w1
   // the same network as SCL:
   "DB365_M_UNIT_02_STA_4".M_CODES_UNIT_02_STA_4.M141 := ("DB337_EXTENDED_M_CODE_UNIT_02_STA_4".M_code[141] OR "DB365_M_UNIT_02_STA_4".M_CODES_UNIT_02_STA_4.M141) AND NOT "DB365_M_UNIT_02_STA_4".M_CODES_UNIT_02_STA_4.Ack_M141 AND NOT "DB2120_MPP_ITC_IPC".RESET_FAULTS AND NOT "DB365_M_UNIT_02_STA_4".M_CODES_UNIT_02_STA_4.M_RESET_PULSE;
END_REGION

REGION Network 73: ACKNOWLEDGE M150-ADVANCE KEYENCE SENSOR POSITION CYLINDER (READ-IN DISABLE) / ACKNOWLEDGE M85-LOAD-UNLOAD TRAP DOOR OPEN
   RUNG wire#powerrail
      Contact( "M_ZERO" )
      Coil( "DB365_M_UNIT_02_STA_4".M_CODES_UNIT_02_STA_4.Ack_M150 )
   END_RUNG
   // the same network as SCL:
   "DB365_M_UNIT_02_STA_4".M_CODES_UNIT_02_STA_4.Ack_M150 := "M_ZERO";
END_REGION

REGION Network 74: M150-ADVANCE KEYENCE SENSOR POSITION CYLINDER (READ-IN DISABLE) / M85-LOAD-UNLOAD TRAP DOOR OPEN
   RUNG wire#powerrail
      Contact( "DB337_EXTENDED_M_CODE_UNIT_02_STA_4".M_code[150] )
      wire#w1
      I_Contact( "DB365_M_UNIT_02_STA_4".M_CODES_UNIT_02_STA_4.Ack_M150 )
      I_Contact( "DB2120_MPP_ITC_IPC".RESET_FAULTS )
      I_Contact( "DB365_M_UNIT_02_STA_4".M_CODES_UNIT_02_STA_4.M_RESET_PULSE )
      Coil( "DB365_M_UNIT_02_STA_4".M_CODES_UNIT_02_STA_4.M150 )
   END_RUNG
   RUNG wire#powerrail
      Contact( "DB365_M_UNIT_02_STA_4".M_CODES_UNIT_02_STA_4.M150 )
   END_RUNG wire#w1
   // the same network as SCL:
   "DB365_M_UNIT_02_STA_4".M_CODES_UNIT_02_STA_4.M150 := ("DB337_EXTENDED_M_CODE_UNIT_02_STA_4".M_code[150] OR "DB365_M_UNIT_02_STA_4".M_CODES_UNIT_02_STA_4.M150) AND NOT "DB365_M_UNIT_02_STA_4".M_CODES_UNIT_02_STA_4.Ack_M150 AND NOT "DB2120_MPP_ITC_IPC".RESET_FAULTS AND NOT "DB365_M_UNIT_02_STA_4".M_CODES_UNIT_02_STA_4.M_RESET_PULSE;
END_REGION

REGION Network 75: ACKNOWLEDGE M151-RETURN KEYENCE SENSOR POSITION CYLINDER (READ-IN DISABLE) / ACKNOWLEDGE M86-LOAD-UNLOAD TRAP DOOR CLOSE
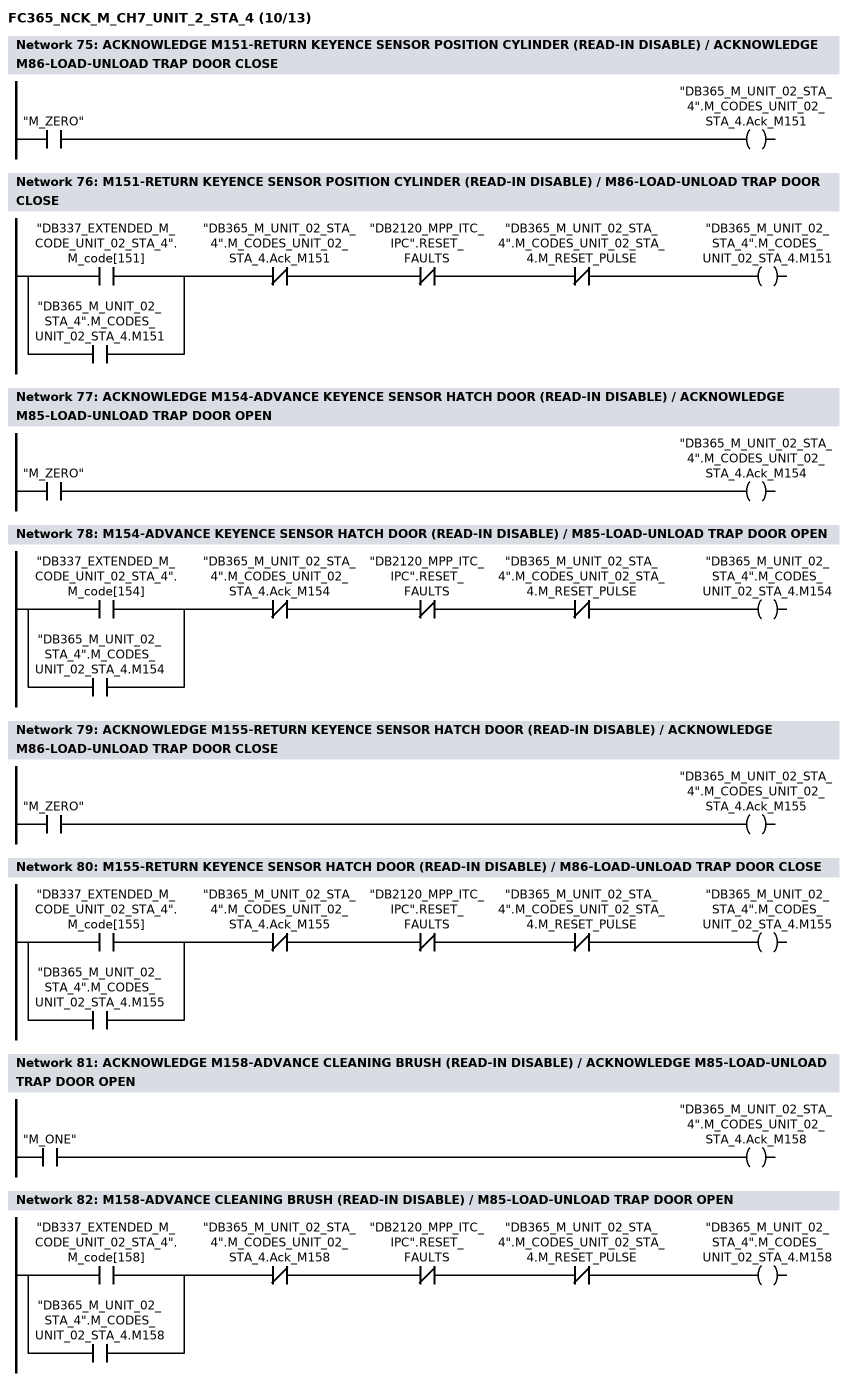
   RUNG wire#powerrail
      Contact( "M_ZERO" )
      Coil( "DB365_M_UNIT_02_STA_4".M_CODES_UNIT_02_STA_4.Ack_M151 )
   END_RUNG
   // the same network as SCL:
   "DB365_M_UNIT_02_STA_4".M_CODES_UNIT_02_STA_4.Ack_M151 := "M_ZERO";
END_REGION

REGION Network 76: M151-RETURN KEYENCE SENSOR POSITION CYLINDER (READ-IN DISABLE) / M86-LOAD-UNLOAD TRAP DOOR CLOSE
   RUNG wire#powerrail
      Contact( "DB337_EXTENDED_M_CODE_UNIT_02_STA_4".M_code[151] )
      wire#w1
      I_Contact( "DB365_M_UNIT_02_STA_4".M_CODES_UNIT_02_STA_4.Ack_M151 )
      I_Contact( "DB2120_MPP_ITC_IPC".RESET_FAULTS )
      I_Contact( "DB365_M_UNIT_02_STA_4".M_CODES_UNIT_02_STA_4.M_RESET_PULSE )
      Coil( "DB365_M_UNIT_02_STA_4".M_CODES_UNIT_02_STA_4.M151 )
   END_RUNG
   RUNG wire#powerrail
      Contact( "DB365_M_UNIT_02_STA_4".M_CODES_UNIT_02_STA_4.M151 )
   END_RUNG wire#w1
   // the same network as SCL:
   "DB365_M_UNIT_02_STA_4".M_CODES_UNIT_02_STA_4.M151 := ("DB337_EXTENDED_M_CODE_UNIT_02_STA_4".M_code[151] OR "DB365_M_UNIT_02_STA_4".M_CODES_UNIT_02_STA_4.M151) AND NOT "DB365_M_UNIT_02_STA_4".M_CODES_UNIT_02_STA_4.Ack_M151 AND NOT "DB2120_MPP_ITC_IPC".RESET_FAULTS AND NOT "DB365_M_UNIT_02_STA_4".M_CODES_UNIT_02_STA_4.M_RESET_PULSE;
END_REGION

REGION Network 77: ACKNOWLEDGE M154-ADVANCE KEYENCE SENSOR HATCH DOOR (READ-IN DISABLE) / ACKNOWLEDGE M85-LOAD-UNLOAD TRAP DOOR OPEN
   RUNG wire#powerrail
      Contact( "M_ZERO" )
      Coil( "DB365_M_UNIT_02_STA_4".M_CODES_UNIT_02_STA_4.Ack_M154 )
   END_RUNG
   // the same network as SCL:
   "DB365_M_UNIT_02_STA_4".M_CODES_UNIT_02_STA_4.Ack_M154 := "M_ZERO";
END_REGION

REGION Network 78: M154-ADVANCE KEYENCE SENSOR HATCH DOOR (READ-IN DISABLE) / M85-LOAD-UNLOAD TRAP DOOR OPEN
   RUNG wire#powerrail
      Contact( "DB337_EXTENDED_M_CODE_UNIT_02_STA_4".M_code[154] )
      wire#w1
      I_Contact( "DB365_M_UNIT_02_STA_4".M_CODES_UNIT_02_STA_4.Ack_M154 )
      I_Contact( "DB2120_MPP_ITC_IPC".RESET_FAULTS )
      I_Contact( "DB365_M_UNIT_02_STA_4".M_CODES_UNIT_02_STA_4.M_RESET_PULSE )
      Coil( "DB365_M_UNIT_02_STA_4".M_CODES_UNIT_02_STA_4.M154 )
   END_RUNG
   RUNG wire#powerrail
      Contact( "DB365_M_UNIT_02_STA_4".M_CODES_UNIT_02_STA_4.M154 )
   END_RUNG wire#w1
   // the same network as SCL:
   "DB365_M_UNIT_02_STA_4".M_CODES_UNIT_02_STA_4.M154 := ("DB337_EXTENDED_M_CODE_UNIT_02_STA_4".M_code[154] OR "DB365_M_UNIT_02_STA_4".M_CODES_UNIT_02_STA_4.M154) AND NOT "DB365_M_UNIT_02_STA_4".M_CODES_UNIT_02_STA_4.Ack_M154 AND NOT "DB2120_MPP_ITC_IPC".RESET_FAULTS AND NOT "DB365_M_UNIT_02_STA_4".M_CODES_UNIT_02_STA_4.M_RESET_PULSE;
END_REGION

REGION Network 79: ACKNOWLEDGE M155-RETURN KEYENCE SENSOR HATCH DOOR (READ-IN DISABLE) / ACKNOWLEDGE M86-LOAD-UNLOAD TRAP DOOR CLOSE
   RUNG wire#powerrail
      Contact( "M_ZERO" )
      Coil( "DB365_M_UNIT_02_STA_4".M_CODES_UNIT_02_STA_4.Ack_M155 )
   END_RUNG
   // the same network as SCL:
   "DB365_M_UNIT_02_STA_4".M_CODES_UNIT_02_STA_4.Ack_M155 := "M_ZERO";
END_REGION

REGION Network 80: M155-RETURN KEYENCE SENSOR HATCH DOOR (READ-IN DISABLE) / M86-LOAD-UNLOAD TRAP DOOR CLOSE
   RUNG wire#powerrail
      Contact( "DB337_EXTENDED_M_CODE_UNIT_02_STA_4".M_code[155] )
      wire#w1
      I_Contact( "DB365_M_UNIT_02_STA_4".M_CODES_UNIT_02_STA_4.Ack_M155 )
      I_Contact( "DB2120_MPP_ITC_IPC".RESET_FAULTS )
      I_Contact( "DB365_M_UNIT_02_STA_4".M_CODES_UNIT_02_STA_4.M_RESET_PULSE )
      Coil( "DB365_M_UNIT_02_STA_4".M_CODES_UNIT_02_STA_4.M155 )
   END_RUNG
   RUNG wire#powerrail
      Contact( "DB365_M_UNIT_02_STA_4".M_CODES_UNIT_02_STA_4.M155 )
   END_RUNG wire#w1
   // the same network as SCL:
   "DB365_M_UNIT_02_STA_4".M_CODES_UNIT_02_STA_4.M155 := ("DB337_EXTENDED_M_CODE_UNIT_02_STA_4".M_code[155] OR "DB365_M_UNIT_02_STA_4".M_CODES_UNIT_02_STA_4.M155) AND NOT "DB365_M_UNIT_02_STA_4".M_CODES_UNIT_02_STA_4.Ack_M155 AND NOT "DB2120_MPP_ITC_IPC".RESET_FAULTS AND NOT "DB365_M_UNIT_02_STA_4".M_CODES_UNIT_02_STA_4.M_RESET_PULSE;
END_REGION

REGION Network 81: ACKNOWLEDGE M158-ADVANCE CLEANING BRUSH (READ-IN DISABLE) / ACKNOWLEDGE M85-LOAD-UNLOAD TRAP DOOR OPEN
   RUNG wire#powerrail
      Contact( "M_ONE" )
      Coil( "DB365_M_UNIT_02_STA_4".M_CODES_UNIT_02_STA_4.Ack_M158 )
   END_RUNG
   // the same network as SCL:
   "DB365_M_UNIT_02_STA_4".M_CODES_UNIT_02_STA_4.Ack_M158 := "M_ONE";
END_REGION

REGION Network 82: M158-ADVANCE CLEANING BRUSH (READ-IN DISABLE) / M85-LOAD-UNLOAD TRAP DOOR OPEN
   RUNG wire#powerrail
      Contact( "DB337_EXTENDED_M_CODE_UNIT_02_STA_4".M_code[158] )
      wire#w1
      I_Contact( "DB365_M_UNIT_02_STA_4".M_CODES_UNIT_02_STA_4.Ack_M158 )
      I_Contact( "DB2120_MPP_ITC_IPC".RESET_FAULTS )
      I_Contact( "DB365_M_UNIT_02_STA_4".M_CODES_UNIT_02_STA_4.M_RESET_PULSE )
      Coil( "DB365_M_UNIT_02_STA_4".M_CODES_UNIT_02_STA_4.M158 )
   END_RUNG
   RUNG wire#powerrail
      Contact( "DB365_M_UNIT_02_STA_4".M_CODES_UNIT_02_STA_4.M158 )
   END_RUNG wire#w1
   // the same network as SCL:
   "DB365_M_UNIT_02_STA_4".M_CODES_UNIT_02_STA_4.M158 := ("DB337_EXTENDED_M_CODE_UNIT_02_STA_4".M_code[158] OR "DB365_M_UNIT_02_STA_4".M_CODES_UNIT_02_STA_4.M158) AND NOT "DB365_M_UNIT_02_STA_4".M_CODES_UNIT_02_STA_4.Ack_M158 AND NOT "DB2120_MPP_ITC_IPC".RESET_FAULTS AND NOT "DB365_M_UNIT_02_STA_4".M_CODES_UNIT_02_STA_4.M_RESET_PULSE;
END_REGION

REGION Network 83: ACKNOWLEDGE M159-RETURN CLEANING BRUSH (READ-IN DISABLE) / ACKNOWLEDGE M86-LOAD-UNLOAD TRAP DOOR CLOSE
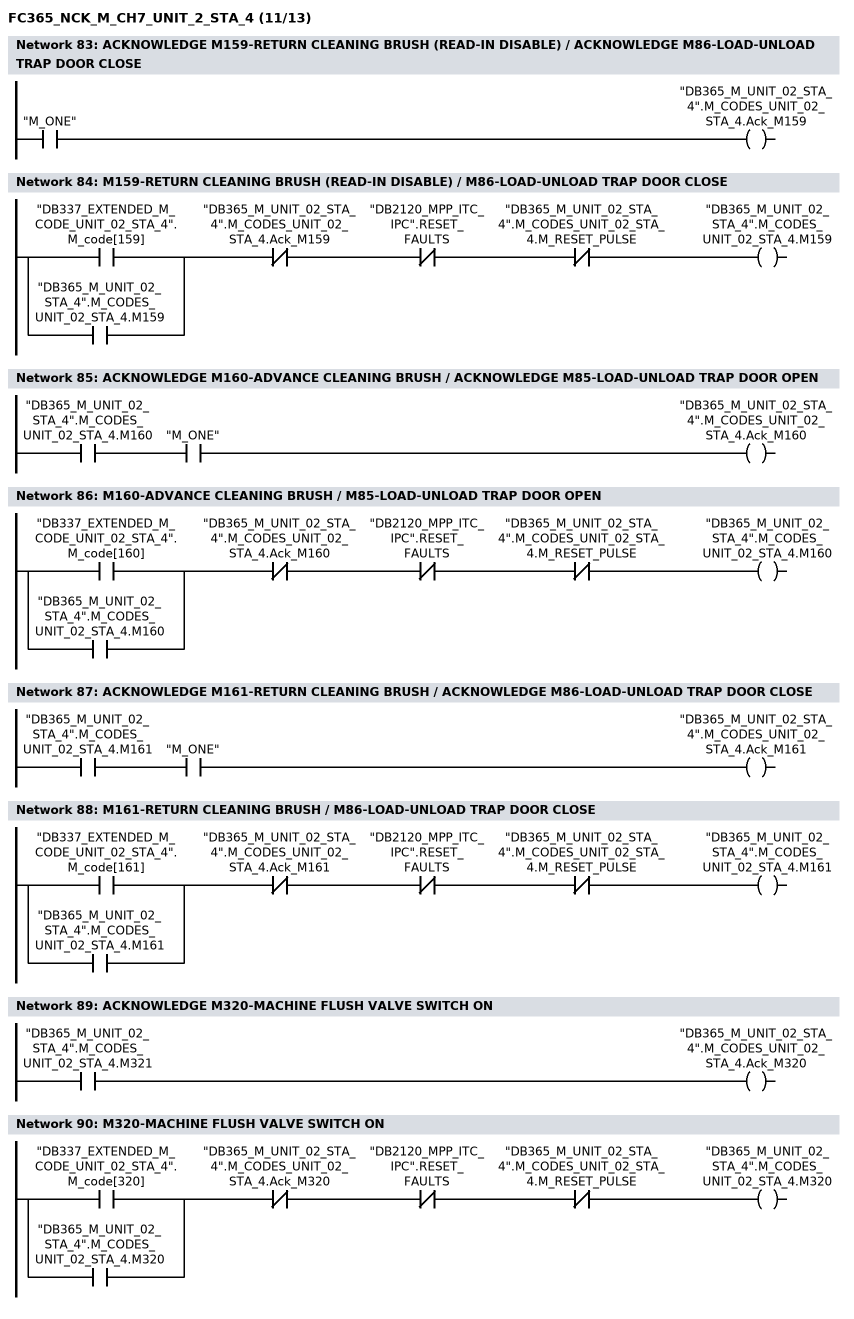
   RUNG wire#powerrail
      Contact( "M_ONE" )
      Coil( "DB365_M_UNIT_02_STA_4".M_CODES_UNIT_02_STA_4.Ack_M159 )
   END_RUNG
   // the same network as SCL:
   "DB365_M_UNIT_02_STA_4".M_CODES_UNIT_02_STA_4.Ack_M159 := "M_ONE";
END_REGION

REGION Network 84: M159-RETURN CLEANING BRUSH (READ-IN DISABLE) / M86-LOAD-UNLOAD TRAP DOOR CLOSE
   RUNG wire#powerrail
      Contact( "DB337_EXTENDED_M_CODE_UNIT_02_STA_4".M_code[159] )
      wire#w1
      I_Contact( "DB365_M_UNIT_02_STA_4".M_CODES_UNIT_02_STA_4.Ack_M159 )
      I_Contact( "DB2120_MPP_ITC_IPC".RESET_FAULTS )
      I_Contact( "DB365_M_UNIT_02_STA_4".M_CODES_UNIT_02_STA_4.M_RESET_PULSE )
      Coil( "DB365_M_UNIT_02_STA_4".M_CODES_UNIT_02_STA_4.M159 )
   END_RUNG
   RUNG wire#powerrail
      Contact( "DB365_M_UNIT_02_STA_4".M_CODES_UNIT_02_STA_4.M159 )
   END_RUNG wire#w1
   // the same network as SCL:
   "DB365_M_UNIT_02_STA_4".M_CODES_UNIT_02_STA_4.M159 := ("DB337_EXTENDED_M_CODE_UNIT_02_STA_4".M_code[159] OR "DB365_M_UNIT_02_STA_4".M_CODES_UNIT_02_STA_4.M159) AND NOT "DB365_M_UNIT_02_STA_4".M_CODES_UNIT_02_STA_4.Ack_M159 AND NOT "DB2120_MPP_ITC_IPC".RESET_FAULTS AND NOT "DB365_M_UNIT_02_STA_4".M_CODES_UNIT_02_STA_4.M_RESET_PULSE;
END_REGION

REGION Network 85: ACKNOWLEDGE M160-ADVANCE CLEANING BRUSH / ACKNOWLEDGE M85-LOAD-UNLOAD TRAP DOOR OPEN
   RUNG wire#powerrail
      Contact( "DB365_M_UNIT_02_STA_4".M_CODES_UNIT_02_STA_4.M160 )
      Contact( "M_ONE" )
      Coil( "DB365_M_UNIT_02_STA_4".M_CODES_UNIT_02_STA_4.Ack_M160 )
   END_RUNG
   // the same network as SCL:
   "DB365_M_UNIT_02_STA_4".M_CODES_UNIT_02_STA_4.Ack_M160 := "DB365_M_UNIT_02_STA_4".M_CODES_UNIT_02_STA_4.M160 AND "M_ONE";
END_REGION

REGION Network 86: M160-ADVANCE CLEANING BRUSH / M85-LOAD-UNLOAD TRAP DOOR OPEN
   RUNG wire#powerrail
      Contact( "DB337_EXTENDED_M_CODE_UNIT_02_STA_4".M_code[160] )
      wire#w1
      I_Contact( "DB365_M_UNIT_02_STA_4".M_CODES_UNIT_02_STA_4.Ack_M160 )
      I_Contact( "DB2120_MPP_ITC_IPC".RESET_FAULTS )
      I_Contact( "DB365_M_UNIT_02_STA_4".M_CODES_UNIT_02_STA_4.M_RESET_PULSE )
      Coil( "DB365_M_UNIT_02_STA_4".M_CODES_UNIT_02_STA_4.M160 )
   END_RUNG
   RUNG wire#powerrail
      Contact( "DB365_M_UNIT_02_STA_4".M_CODES_UNIT_02_STA_4.M160 )
   END_RUNG wire#w1
   // the same network as SCL:
   "DB365_M_UNIT_02_STA_4".M_CODES_UNIT_02_STA_4.M160 := ("DB337_EXTENDED_M_CODE_UNIT_02_STA_4".M_code[160] OR "DB365_M_UNIT_02_STA_4".M_CODES_UNIT_02_STA_4.M160) AND NOT "DB365_M_UNIT_02_STA_4".M_CODES_UNIT_02_STA_4.Ack_M160 AND NOT "DB2120_MPP_ITC_IPC".RESET_FAULTS AND NOT "DB365_M_UNIT_02_STA_4".M_CODES_UNIT_02_STA_4.M_RESET_PULSE;
END_REGION

REGION Network 87: ACKNOWLEDGE M161-RETURN CLEANING BRUSH / ACKNOWLEDGE M86-LOAD-UNLOAD TRAP DOOR CLOSE
   RUNG wire#powerrail
      Contact( "DB365_M_UNIT_02_STA_4".M_CODES_UNIT_02_STA_4.M161 )
      Contact( "M_ONE" )
      Coil( "DB365_M_UNIT_02_STA_4".M_CODES_UNIT_02_STA_4.Ack_M161 )
   END_RUNG
   // the same network as SCL:
   "DB365_M_UNIT_02_STA_4".M_CODES_UNIT_02_STA_4.Ack_M161 := "DB365_M_UNIT_02_STA_4".M_CODES_UNIT_02_STA_4.M161 AND "M_ONE";
END_REGION

REGION Network 88: M161-RETURN CLEANING BRUSH / M86-LOAD-UNLOAD TRAP DOOR CLOSE
   RUNG wire#powerrail
      Contact( "DB337_EXTENDED_M_CODE_UNIT_02_STA_4".M_code[161] )
      wire#w1
      I_Contact( "DB365_M_UNIT_02_STA_4".M_CODES_UNIT_02_STA_4.Ack_M161 )
      I_Contact( "DB2120_MPP_ITC_IPC".RESET_FAULTS )
      I_Contact( "DB365_M_UNIT_02_STA_4".M_CODES_UNIT_02_STA_4.M_RESET_PULSE )
      Coil( "DB365_M_UNIT_02_STA_4".M_CODES_UNIT_02_STA_4.M161 )
   END_RUNG
   RUNG wire#powerrail
      Contact( "DB365_M_UNIT_02_STA_4".M_CODES_UNIT_02_STA_4.M161 )
   END_RUNG wire#w1
   // the same network as SCL:
   "DB365_M_UNIT_02_STA_4".M_CODES_UNIT_02_STA_4.M161 := ("DB337_EXTENDED_M_CODE_UNIT_02_STA_4".M_code[161] OR "DB365_M_UNIT_02_STA_4".M_CODES_UNIT_02_STA_4.M161) AND NOT "DB365_M_UNIT_02_STA_4".M_CODES_UNIT_02_STA_4.Ack_M161 AND NOT "DB2120_MPP_ITC_IPC".RESET_FAULTS AND NOT "DB365_M_UNIT_02_STA_4".M_CODES_UNIT_02_STA_4.M_RESET_PULSE;
END_REGION

REGION Network 89: ACKNOWLEDGE M320-MACHINE FLUSH VALVE SWITCH ON
   RUNG wire#powerrail
      Contact( "DB365_M_UNIT_02_STA_4".M_CODES_UNIT_02_STA_4.M321 )
      Coil( "DB365_M_UNIT_02_STA_4".M_CODES_UNIT_02_STA_4.Ack_M320 )
   END_RUNG
   // the same network as SCL:
   "DB365_M_UNIT_02_STA_4".M_CODES_UNIT_02_STA_4.Ack_M320 := "DB365_M_UNIT_02_STA_4".M_CODES_UNIT_02_STA_4.M321;
END_REGION

REGION Network 90: M320-MACHINE FLUSH VALVE SWITCH ON
   RUNG wire#powerrail
      Contact( "DB337_EXTENDED_M_CODE_UNIT_02_STA_4".M_code[320] )
      wire#w1
      I_Contact( "DB365_M_UNIT_02_STA_4".M_CODES_UNIT_02_STA_4.Ack_M320 )
      I_Contact( "DB2120_MPP_ITC_IPC".RESET_FAULTS )
      I_Contact( "DB365_M_UNIT_02_STA_4".M_CODES_UNIT_02_STA_4.M_RESET_PULSE )
      Coil( "DB365_M_UNIT_02_STA_4".M_CODES_UNIT_02_STA_4.M320 )
   END_RUNG
   RUNG wire#powerrail
      Contact( "DB365_M_UNIT_02_STA_4".M_CODES_UNIT_02_STA_4.M320 )
   END_RUNG wire#w1
   // the same network as SCL:
   "DB365_M_UNIT_02_STA_4".M_CODES_UNIT_02_STA_4.M320 := ("DB337_EXTENDED_M_CODE_UNIT_02_STA_4".M_code[320] OR "DB365_M_UNIT_02_STA_4".M_CODES_UNIT_02_STA_4.M320) AND NOT "DB365_M_UNIT_02_STA_4".M_CODES_UNIT_02_STA_4.Ack_M320 AND NOT "DB2120_MPP_ITC_IPC".RESET_FAULTS AND NOT "DB365_M_UNIT_02_STA_4".M_CODES_UNIT_02_STA_4.M_RESET_PULSE;
END_REGION

REGION Network 91: ACKNOWLEDGE M321-MACHINE FLUSH VALVE SWITCH OFF
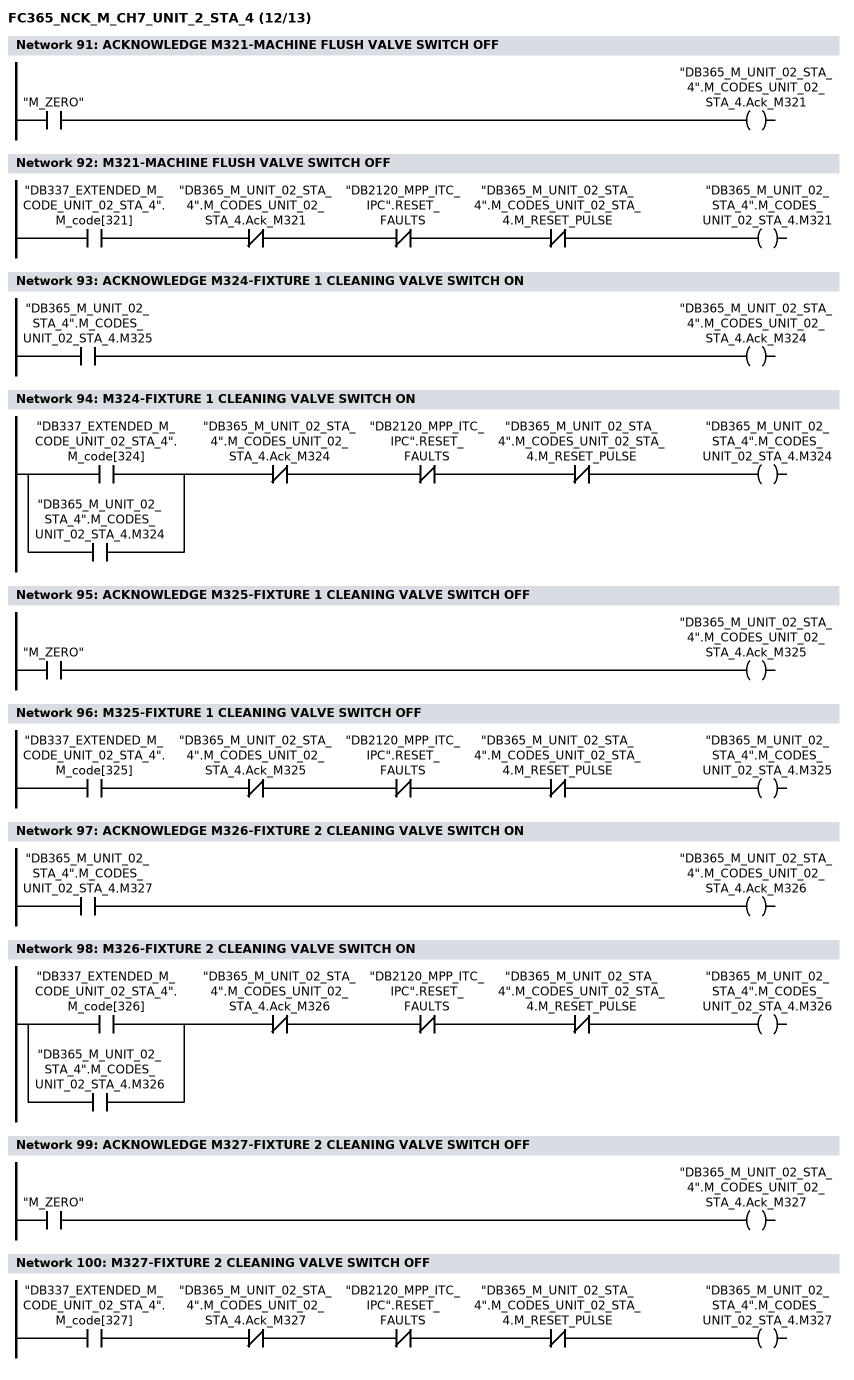
   RUNG wire#powerrail
      Contact( "M_ZERO" )
      Coil( "DB365_M_UNIT_02_STA_4".M_CODES_UNIT_02_STA_4.Ack_M321 )
   END_RUNG
   // the same network as SCL:
   "DB365_M_UNIT_02_STA_4".M_CODES_UNIT_02_STA_4.Ack_M321 := "M_ZERO";
END_REGION

REGION Network 92: M321-MACHINE FLUSH VALVE SWITCH OFF
   RUNG wire#powerrail
      Contact( "DB337_EXTENDED_M_CODE_UNIT_02_STA_4".M_code[321] )
      I_Contact( "DB365_M_UNIT_02_STA_4".M_CODES_UNIT_02_STA_4.Ack_M321 )
      I_Contact( "DB2120_MPP_ITC_IPC".RESET_FAULTS )
      I_Contact( "DB365_M_UNIT_02_STA_4".M_CODES_UNIT_02_STA_4.M_RESET_PULSE )
      Coil( "DB365_M_UNIT_02_STA_4".M_CODES_UNIT_02_STA_4.M321 )
   END_RUNG
   // the same network as SCL:
   "DB365_M_UNIT_02_STA_4".M_CODES_UNIT_02_STA_4.M321 := "DB337_EXTENDED_M_CODE_UNIT_02_STA_4".M_code[321] AND NOT "DB365_M_UNIT_02_STA_4".M_CODES_UNIT_02_STA_4.Ack_M321 AND NOT "DB2120_MPP_ITC_IPC".RESET_FAULTS AND NOT "DB365_M_UNIT_02_STA_4".M_CODES_UNIT_02_STA_4.M_RESET_PULSE;
END_REGION

REGION Network 93: ACKNOWLEDGE M324-FIXTURE 1 CLEANING VALVE SWITCH ON
   RUNG wire#powerrail
      Contact( "DB365_M_UNIT_02_STA_4".M_CODES_UNIT_02_STA_4.M325 )
      Coil( "DB365_M_UNIT_02_STA_4".M_CODES_UNIT_02_STA_4.Ack_M324 )
   END_RUNG
   // the same network as SCL:
   "DB365_M_UNIT_02_STA_4".M_CODES_UNIT_02_STA_4.Ack_M324 := "DB365_M_UNIT_02_STA_4".M_CODES_UNIT_02_STA_4.M325;
END_REGION

REGION Network 94: M324-FIXTURE 1 CLEANING VALVE SWITCH ON
   RUNG wire#powerrail
      Contact( "DB337_EXTENDED_M_CODE_UNIT_02_STA_4".M_code[324] )
      wire#w1
      I_Contact( "DB365_M_UNIT_02_STA_4".M_CODES_UNIT_02_STA_4.Ack_M324 )
      I_Contact( "DB2120_MPP_ITC_IPC".RESET_FAULTS )
      I_Contact( "DB365_M_UNIT_02_STA_4".M_CODES_UNIT_02_STA_4.M_RESET_PULSE )
      Coil( "DB365_M_UNIT_02_STA_4".M_CODES_UNIT_02_STA_4.M324 )
   END_RUNG
   RUNG wire#powerrail
      Contact( "DB365_M_UNIT_02_STA_4".M_CODES_UNIT_02_STA_4.M324 )
   END_RUNG wire#w1
   // the same network as SCL:
   "DB365_M_UNIT_02_STA_4".M_CODES_UNIT_02_STA_4.M324 := ("DB337_EXTENDED_M_CODE_UNIT_02_STA_4".M_code[324] OR "DB365_M_UNIT_02_STA_4".M_CODES_UNIT_02_STA_4.M324) AND NOT "DB365_M_UNIT_02_STA_4".M_CODES_UNIT_02_STA_4.Ack_M324 AND NOT "DB2120_MPP_ITC_IPC".RESET_FAULTS AND NOT "DB365_M_UNIT_02_STA_4".M_CODES_UNIT_02_STA_4.M_RESET_PULSE;
END_REGION

REGION Network 95: ACKNOWLEDGE M325-FIXTURE 1 CLEANING VALVE SWITCH OFF
   RUNG wire#powerrail
      Contact( "M_ZERO" )
      Coil( "DB365_M_UNIT_02_STA_4".M_CODES_UNIT_02_STA_4.Ack_M325 )
   END_RUNG
   // the same network as SCL:
   "DB365_M_UNIT_02_STA_4".M_CODES_UNIT_02_STA_4.Ack_M325 := "M_ZERO";
END_REGION

REGION Network 96: M325-FIXTURE 1 CLEANING VALVE SWITCH OFF
   RUNG wire#powerrail
      Contact( "DB337_EXTENDED_M_CODE_UNIT_02_STA_4".M_code[325] )
      I_Contact( "DB365_M_UNIT_02_STA_4".M_CODES_UNIT_02_STA_4.Ack_M325 )
      I_Contact( "DB2120_MPP_ITC_IPC".RESET_FAULTS )
      I_Contact( "DB365_M_UNIT_02_STA_4".M_CODES_UNIT_02_STA_4.M_RESET_PULSE )
      Coil( "DB365_M_UNIT_02_STA_4".M_CODES_UNIT_02_STA_4.M325 )
   END_RUNG
   // the same network as SCL:
   "DB365_M_UNIT_02_STA_4".M_CODES_UNIT_02_STA_4.M325 := "DB337_EXTENDED_M_CODE_UNIT_02_STA_4".M_code[325] AND NOT "DB365_M_UNIT_02_STA_4".M_CODES_UNIT_02_STA_4.Ack_M325 AND NOT "DB2120_MPP_ITC_IPC".RESET_FAULTS AND NOT "DB365_M_UNIT_02_STA_4".M_CODES_UNIT_02_STA_4.M_RESET_PULSE;
END_REGION

REGION Network 97: ACKNOWLEDGE M326-FIXTURE 2 CLEANING VALVE SWITCH ON
   RUNG wire#powerrail
      Contact( "DB365_M_UNIT_02_STA_4".M_CODES_UNIT_02_STA_4.M327 )
      Coil( "DB365_M_UNIT_02_STA_4".M_CODES_UNIT_02_STA_4.Ack_M326 )
   END_RUNG
   // the same network as SCL:
   "DB365_M_UNIT_02_STA_4".M_CODES_UNIT_02_STA_4.Ack_M326 := "DB365_M_UNIT_02_STA_4".M_CODES_UNIT_02_STA_4.M327;
END_REGION

REGION Network 98: M326-FIXTURE 2 CLEANING VALVE SWITCH ON
   RUNG wire#powerrail
      Contact( "DB337_EXTENDED_M_CODE_UNIT_02_STA_4".M_code[326] )
      wire#w1
      I_Contact( "DB365_M_UNIT_02_STA_4".M_CODES_UNIT_02_STA_4.Ack_M326 )
      I_Contact( "DB2120_MPP_ITC_IPC".RESET_FAULTS )
      I_Contact( "DB365_M_UNIT_02_STA_4".M_CODES_UNIT_02_STA_4.M_RESET_PULSE )
      Coil( "DB365_M_UNIT_02_STA_4".M_CODES_UNIT_02_STA_4.M326 )
   END_RUNG
   RUNG wire#powerrail
      Contact( "DB365_M_UNIT_02_STA_4".M_CODES_UNIT_02_STA_4.M326 )
   END_RUNG wire#w1
   // the same network as SCL:
   "DB365_M_UNIT_02_STA_4".M_CODES_UNIT_02_STA_4.M326 := ("DB337_EXTENDED_M_CODE_UNIT_02_STA_4".M_code[326] OR "DB365_M_UNIT_02_STA_4".M_CODES_UNIT_02_STA_4.M326) AND NOT "DB365_M_UNIT_02_STA_4".M_CODES_UNIT_02_STA_4.Ack_M326 AND NOT "DB2120_MPP_ITC_IPC".RESET_FAULTS AND NOT "DB365_M_UNIT_02_STA_4".M_CODES_UNIT_02_STA_4.M_RESET_PULSE;
END_REGION

REGION Network 99: ACKNOWLEDGE M327-FIXTURE 2 CLEANING VALVE SWITCH OFF
   RUNG wire#powerrail
      Contact( "M_ZERO" )
      Coil( "DB365_M_UNIT_02_STA_4".M_CODES_UNIT_02_STA_4.Ack_M327 )
   END_RUNG
   // the same network as SCL:
   "DB365_M_UNIT_02_STA_4".M_CODES_UNIT_02_STA_4.Ack_M327 := "M_ZERO";
END_REGION

REGION Network 100: M327-FIXTURE 2 CLEANING VALVE SWITCH OFF
   RUNG wire#powerrail
      Contact( "DB337_EXTENDED_M_CODE_UNIT_02_STA_4".M_code[327] )
      I_Contact( "DB365_M_UNIT_02_STA_4".M_CODES_UNIT_02_STA_4.Ack_M327 )
      I_Contact( "DB2120_MPP_ITC_IPC".RESET_FAULTS )
      I_Contact( "DB365_M_UNIT_02_STA_4".M_CODES_UNIT_02_STA_4.M_RESET_PULSE )
      Coil( "DB365_M_UNIT_02_STA_4".M_CODES_UNIT_02_STA_4.M327 )
   END_RUNG
   // the same network as SCL:
   "DB365_M_UNIT_02_STA_4".M_CODES_UNIT_02_STA_4.M327 := "DB337_EXTENDED_M_CODE_UNIT_02_STA_4".M_code[327] AND NOT "DB365_M_UNIT_02_STA_4".M_CODES_UNIT_02_STA_4.Ack_M327 AND NOT "DB2120_MPP_ITC_IPC".RESET_FAULTS AND NOT "DB365_M_UNIT_02_STA_4".M_CODES_UNIT_02_STA_4.M_RESET_PULSE;
END_REGION

REGION Network 101: ACKNOWLEDGE M332-FIXTURE 1 INTERNAL BLOWING SWITCH ON
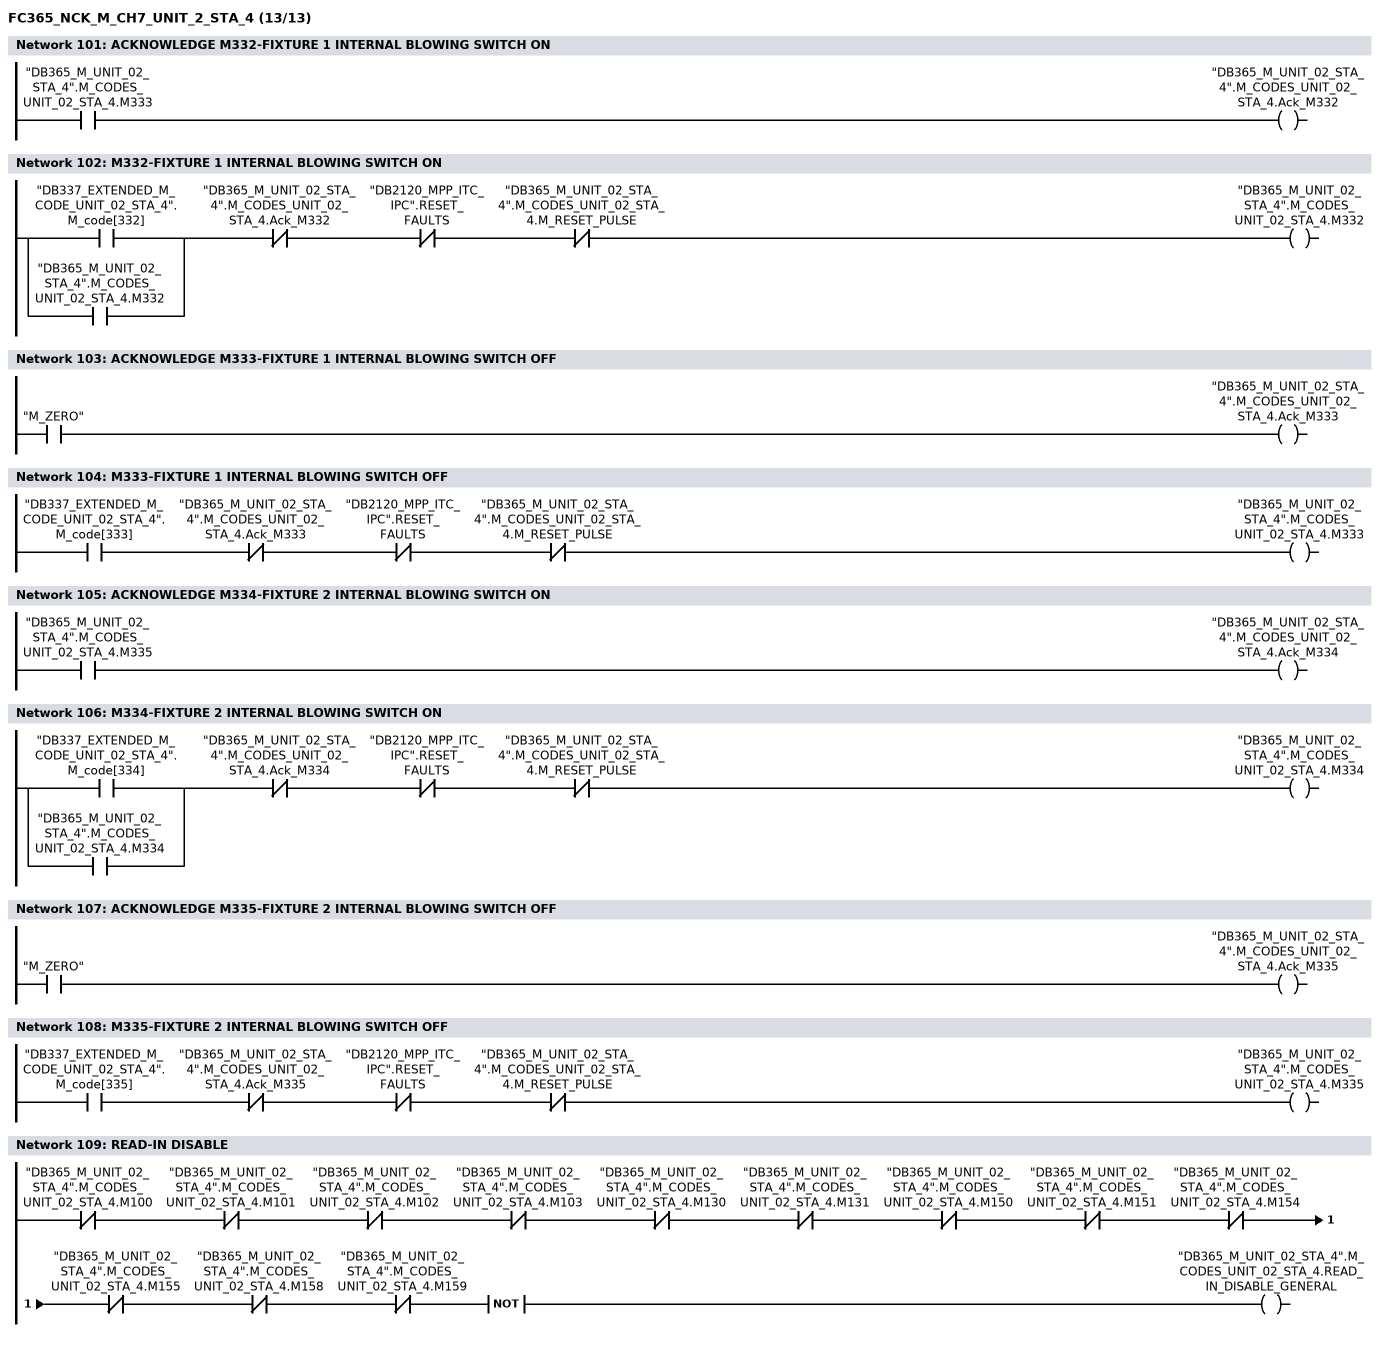
   RUNG wire#powerrail
      Contact( "DB365_M_UNIT_02_STA_4".M_CODES_UNIT_02_STA_4.M333 )
      Coil( "DB365_M_UNIT_02_STA_4".M_CODES_UNIT_02_STA_4.Ack_M332 )
   END_RUNG
   // the same network as SCL:
   "DB365_M_UNIT_02_STA_4".M_CODES_UNIT_02_STA_4.Ack_M332 := "DB365_M_UNIT_02_STA_4".M_CODES_UNIT_02_STA_4.M333;
END_REGION

REGION Network 102: M332-FIXTURE 1 INTERNAL BLOWING SWITCH ON
   RUNG wire#powerrail
      Contact( "DB337_EXTENDED_M_CODE_UNIT_02_STA_4".M_code[332] )
      wire#w1
      I_Contact( "DB365_M_UNIT_02_STA_4".M_CODES_UNIT_02_STA_4.Ack_M332 )
      I_Contact( "DB2120_MPP_ITC_IPC".RESET_FAULTS )
      I_Contact( "DB365_M_UNIT_02_STA_4".M_CODES_UNIT_02_STA_4.M_RESET_PULSE )
      Coil( "DB365_M_UNIT_02_STA_4".M_CODES_UNIT_02_STA_4.M332 )
   END_RUNG
   RUNG wire#powerrail
      Contact( "DB365_M_UNIT_02_STA_4".M_CODES_UNIT_02_STA_4.M332 )
   END_RUNG wire#w1
   // the same network as SCL:
   "DB365_M_UNIT_02_STA_4".M_CODES_UNIT_02_STA_4.M332 := ("DB337_EXTENDED_M_CODE_UNIT_02_STA_4".M_code[332] OR "DB365_M_UNIT_02_STA_4".M_CODES_UNIT_02_STA_4.M332) AND NOT "DB365_M_UNIT_02_STA_4".M_CODES_UNIT_02_STA_4.Ack_M332 AND NOT "DB2120_MPP_ITC_IPC".RESET_FAULTS AND NOT "DB365_M_UNIT_02_STA_4".M_CODES_UNIT_02_STA_4.M_RESET_PULSE;
END_REGION

REGION Network 103: ACKNOWLEDGE M333-FIXTURE 1 INTERNAL BLOWING SWITCH OFF
   RUNG wire#powerrail
      Contact( "M_ZERO" )
      Coil( "DB365_M_UNIT_02_STA_4".M_CODES_UNIT_02_STA_4.Ack_M333 )
   END_RUNG
   // the same network as SCL:
   "DB365_M_UNIT_02_STA_4".M_CODES_UNIT_02_STA_4.Ack_M333 := "M_ZERO";
END_REGION

REGION Network 104: M333-FIXTURE 1 INTERNAL BLOWING SWITCH OFF
   RUNG wire#powerrail
      Contact( "DB337_EXTENDED_M_CODE_UNIT_02_STA_4".M_code[333] )
      I_Contact( "DB365_M_UNIT_02_STA_4".M_CODES_UNIT_02_STA_4.Ack_M333 )
      I_Contact( "DB2120_MPP_ITC_IPC".RESET_FAULTS )
      I_Contact( "DB365_M_UNIT_02_STA_4".M_CODES_UNIT_02_STA_4.M_RESET_PULSE )
      Coil( "DB365_M_UNIT_02_STA_4".M_CODES_UNIT_02_STA_4.M333 )
   END_RUNG
   // the same network as SCL:
   "DB365_M_UNIT_02_STA_4".M_CODES_UNIT_02_STA_4.M333 := "DB337_EXTENDED_M_CODE_UNIT_02_STA_4".M_code[333] AND NOT "DB365_M_UNIT_02_STA_4".M_CODES_UNIT_02_STA_4.Ack_M333 AND NOT "DB2120_MPP_ITC_IPC".RESET_FAULTS AND NOT "DB365_M_UNIT_02_STA_4".M_CODES_UNIT_02_STA_4.M_RESET_PULSE;
END_REGION

REGION Network 105: ACKNOWLEDGE M334-FIXTURE 2 INTERNAL BLOWING SWITCH ON
   RUNG wire#powerrail
      Contact( "DB365_M_UNIT_02_STA_4".M_CODES_UNIT_02_STA_4.M335 )
      Coil( "DB365_M_UNIT_02_STA_4".M_CODES_UNIT_02_STA_4.Ack_M334 )
   END_RUNG
   // the same network as SCL:
   "DB365_M_UNIT_02_STA_4".M_CODES_UNIT_02_STA_4.Ack_M334 := "DB365_M_UNIT_02_STA_4".M_CODES_UNIT_02_STA_4.M335;
END_REGION

REGION Network 106: M334-FIXTURE 2 INTERNAL BLOWING SWITCH ON
   RUNG wire#powerrail
      Contact( "DB337_EXTENDED_M_CODE_UNIT_02_STA_4".M_code[334] )
      wire#w1
      I_Contact( "DB365_M_UNIT_02_STA_4".M_CODES_UNIT_02_STA_4.Ack_M334 )
      I_Contact( "DB2120_MPP_ITC_IPC".RESET_FAULTS )
      I_Contact( "DB365_M_UNIT_02_STA_4".M_CODES_UNIT_02_STA_4.M_RESET_PULSE )
      Coil( "DB365_M_UNIT_02_STA_4".M_CODES_UNIT_02_STA_4.M334 )
   END_RUNG
   RUNG wire#powerrail
      Contact( "DB365_M_UNIT_02_STA_4".M_CODES_UNIT_02_STA_4.M334 )
   END_RUNG wire#w1
   // the same network as SCL:
   "DB365_M_UNIT_02_STA_4".M_CODES_UNIT_02_STA_4.M334 := ("DB337_EXTENDED_M_CODE_UNIT_02_STA_4".M_code[334] OR "DB365_M_UNIT_02_STA_4".M_CODES_UNIT_02_STA_4.M334) AND NOT "DB365_M_UNIT_02_STA_4".M_CODES_UNIT_02_STA_4.Ack_M334 AND NOT "DB2120_MPP_ITC_IPC".RESET_FAULTS AND NOT "DB365_M_UNIT_02_STA_4".M_CODES_UNIT_02_STA_4.M_RESET_PULSE;
END_REGION

REGION Network 107: ACKNOWLEDGE M335-FIXTURE 2 INTERNAL BLOWING SWITCH OFF
   RUNG wire#powerrail
      Contact( "M_ZERO" )
      Coil( "DB365_M_UNIT_02_STA_4".M_CODES_UNIT_02_STA_4.Ack_M335 )
   END_RUNG
   // the same network as SCL:
   "DB365_M_UNIT_02_STA_4".M_CODES_UNIT_02_STA_4.Ack_M335 := "M_ZERO";
END_REGION

REGION Network 108: M335-FIXTURE 2 INTERNAL BLOWING SWITCH OFF
   RUNG wire#powerrail
      Contact( "DB337_EXTENDED_M_CODE_UNIT_02_STA_4".M_code[335] )
      I_Contact( "DB365_M_UNIT_02_STA_4".M_CODES_UNIT_02_STA_4.Ack_M335 )
      I_Contact( "DB2120_MPP_ITC_IPC".RESET_FAULTS )
      I_Contact( "DB365_M_UNIT_02_STA_4".M_CODES_UNIT_02_STA_4.M_RESET_PULSE )
      Coil( "DB365_M_UNIT_02_STA_4".M_CODES_UNIT_02_STA_4.M335 )
   END_RUNG
   // the same network as SCL:
   "DB365_M_UNIT_02_STA_4".M_CODES_UNIT_02_STA_4.M335 := "DB337_EXTENDED_M_CODE_UNIT_02_STA_4".M_code[335] AND NOT "DB365_M_UNIT_02_STA_4".M_CODES_UNIT_02_STA_4.Ack_M335 AND NOT "DB2120_MPP_ITC_IPC".RESET_FAULTS AND NOT "DB365_M_UNIT_02_STA_4".M_CODES_UNIT_02_STA_4.M_RESET_PULSE;
END_REGION

REGION Network 109: READ-IN DISABLE
   RUNG wire#powerrail
      I_Contact( "DB365_M_UNIT_02_STA_4".M_CODES_UNIT_02_STA_4.M100 )
      I_Contact( "DB365_M_UNIT_02_STA_4".M_CODES_UNIT_02_STA_4.M101 )
      I_Contact( "DB365_M_UNIT_02_STA_4".M_CODES_UNIT_02_STA_4.M102 )
      I_Contact( "DB365_M_UNIT_02_STA_4".M_CODES_UNIT_02_STA_4.M103 )
      I_Contact( "DB365_M_UNIT_02_STA_4".M_CODES_UNIT_02_STA_4.M130 )
      I_Contact( "DB365_M_UNIT_02_STA_4".M_CODES_UNIT_02_STA_4.M131 )
      I_Contact( "DB365_M_UNIT_02_STA_4".M_CODES_UNIT_02_STA_4.M150 )
      I_Contact( "DB365_M_UNIT_02_STA_4".M_CODES_UNIT_02_STA_4.M151 )
      I_Contact( "DB365_M_UNIT_02_STA_4".M_CODES_UNIT_02_STA_4.M154 )
      I_Contact( "DB365_M_UNIT_02_STA_4".M_CODES_UNIT_02_STA_4.M155 )
      I_Contact( "DB365_M_UNIT_02_STA_4".M_CODES_UNIT_02_STA_4.M158 )
      I_Contact( "DB365_M_UNIT_02_STA_4".M_CODES_UNIT_02_STA_4.M159 )
      Not()
      Coil( "DB365_M_UNIT_02_STA_4".M_CODES_UNIT_02_STA_4.READ_IN_DISABLE_GENERAL )
   END_RUNG
   // the same network as SCL:
   "DB365_M_UNIT_02_STA_4".M_CODES_UNIT_02_STA_4.READ_IN_DISABLE_GENERAL := NOT (NOT "DB365_M_UNIT_02_STA_4".M_CODES_UNIT_02_STA_4.M100 AND NOT "DB365_M_UNIT_02_STA_4".M_CODES_UNIT_02_STA_4.M101 AND NOT "DB365_M_UNIT_02_STA_4".M_CODES_UNIT_02_STA_4.M102 AND NOT "DB365_M_UNIT_02_STA_4".M_CODES_UNIT_02_STA_4.M103 AND NOT "DB365_M_UNIT_02_STA_4".M_CODES_UNIT_02_STA_4.M130 AND NOT "DB365_M_UNIT_02_STA_4".M_CODES_UNIT_02_STA_4.M131 AND NOT "DB365_M_UNIT_02_STA_4".M_CODES_UNIT_02_STA_4.M150 AND NOT "DB365_M_UNIT_02_STA_4".M_CODES_UNIT_02_STA_4.M151 AND NOT "DB365_M_UNIT_02_STA_4".M_CODES_UNIT_02_STA_4.M154 AND NOT "DB365_M_UNIT_02_STA_4".M_CODES_UNIT_02_STA_4.M155 AND NOT "DB365_M_UNIT_02_STA_4".M_CODES_UNIT_02_STA_4.M158 AND NOT "DB365_M_UNIT_02_STA_4".M_CODES_UNIT_02_STA_4.M159);
END_REGION
END_FUNCTION
